C03641=1066.712,243.059,411.910,173.514,30.736,155.609
C03642=1066.719,243.308,411.883,173.516,30.739,155.610
C03643=1066.724,243.556,411.855,173.519,30.744,155.610
C03644=1066.731,243.805,411.827,173.521,30.748,155.611
C03645=1066.736,244.053,411.800,173.523,30.751,155.612
C03646=1066.743,244.302,411.772,173.526,30.756,155.613
C03647=1066.748,244.550,411.744,173.527,30.759,155.613
C03648=1066.754,244.799,411.717,173.530,30.763,155.614
C03649=1066.760,245.047,411.689,173.533,30.768,155.615
C03650=1066.766,245.295,411.661,173.534,30.771,155.615
C03651=1066.772,245.543,411.634,173.537,30.775,155.616
C03652=1066.778,245.792,411.606,173.540,30.780,155.617
C03653=1066.783,246.041,411.579,173.542,30.783,155.617
C03654=1066.790,246.289,411.551,173.544,30.787,155.618
C03655=1066.796,246.538,411.522,173.547,30.792,155.619
C03656=1066.802,246.785,411.495,173.549,30.795,155.619
C03657=1066.808,247.034,411.467,173.551,30.799,155.620
C03658=1066.813,247.283,411.440,173.553,30.804,155.621
C03659=1066.819,247.532,411.411,173.556,30.807,155.622
C03660=1066.825,247.779,411.384,173.558,30.812,155.622
C03661=1066.831,248.028,411.356,173.560,30.815,155.623
C03662=1066.836,248.276,411.328,173.563,30.819,155.624
C03663=1066.843,248.525,411.300,173.566,30.824,155.624
C03664=1066.848,248.740,411.275,173.567,30.827,155.625
C03665=1066.853,248.954,411.252,173.569,30.831,155.626
C03666=1066.858,249.169,411.227,173.572,30.834,155.626
C03667=1066.863,249.384,411.203,173.574,30.838,155.627
C03668=1066.868,249.599,411.179,173.575,30.841,155.627
C03669=1066.873,249.814,411.155,173.577,30.844,155.628
C03670=1066.878,250.029,411.130,173.580,30.848,155.629
C03671=1066.884,250.244,411.106,173.582,30.851,155.629
C03672=1066.889,250.492,411.078,173.584,30.855,155.630
C03673=1066.895,250.740,411.049,173.586,30.859,155.631
C03674=1066.901,250.989,411.021,173.589,30.863,155.631
C03675=1066.907,251.237,410.994,173.591,30.868,155.632
C03676=1066.913,251.485,410.965,173.593,30.871,155.633
C03677=1066.918,251.733,410.937,173.596,30.875,155.634
C03678=1066.924,251.982,410.909,173.599,30.880,155.634
C03679=1066.930,252.231,410.881,173.600,30.883,155.635
C03680=1066.936,252.479,410.853,173.603,30.887,155.636
C03681=1066.942,252.727,410.825,173.606,30.892,155.636
C03682=1066.949,252.976,410.796,173.608,30.896,155.637
C03683=1066.954,253.224,410.768,173.610,30.899,155.638
C03684=1066.961,253.472,410.740,173.613,30.904,155.639
C03685=1066.967,253.721,410.712,173.616,30.907,155.639
C03686=1066.972,253.969,410.684,173.617,30.911,155.640
C03687=1066.978,254.217,410.655,173.620,30.916,155.641
C03688=1066.984,254.466,410.627,173.623,30.919,155.641
C03689=1066.991,254.714,410.599,173.625,30.923,155.642
C03690=1066.996,254.962,410.571,173.627,30.927,155.643
C03691=1067.002,255.210,410.542,173.630,30.931,155.643
C03692=1067.008,255.459,410.514,173.633,30.935,155.644
C03693=1067.014,255.707,410.486,173.634,30.939,155.645
C03694=1067.020,255.955,410.457,173.637,30.943,155.645
C03695=1067.027,256.204,410.429,173.640,30.947,155.646
C03696=1067.033,256.453,410.401,173.642,30.951,155.647
C03697=1067.039,256.701,410.372,173.644,30.955,155.648
C03698=1067.044,256.949,410.344,173.647,30.959,155.648
C03699=1067.050,257.197,410.315,173.650,30.963,155.649
C03700=1067.056,257.446,410.286,173.652,30.967,155.650
C03701=1067.063,257.694,410.258,173.654,30.971,155.650
C03702=1067.069,257.941,410.230,173.657,30.975,155.651
C03703=1067.075,258.190,410.201,173.660,30.979,155.652
C03704=1067.081,258.439,410.173,173.661,30.983,155.652
C03705=1067.087,258.687,410.144,173.664,30.987,155.653
C03706=1067.093,258.936,410.116,173.667,30.991,155.654
C03707=1067.099,259.184,410.087,173.669,30.994,155.654
C03708=1067.104,259.432,410.059,173.672,30.999,155.655
C03709=1067.111,259.680,410.030,173.674,31.002,155.656
C03710=1067.117,259.929,410.002,173.677,31.006,155.657
C03711=1067.124,260.177,409.973,173.679,31.010,155.657
C03712=1067.130,260.425,409.944,173.682,31.015,155.658
C03713=1067.136,260.674,409.916,173.684,31.018,155.659
C03714=1067.142,260.922,409.887,173.687,31.022,155.659
C03715=1067.148,261.171,409.858,173.689,31.026,155.660
C03716=1067.154,261.419,409.829,173.692,31.030,155.661
C03717=1067.160,261.666,409.801,173.695,31.034,155.661
C03718=1067.167,261.914,409.773,173.697,31.038,155.662
C03719=1067.173,262.163,409.744,173.699,31.042,155.663
C03720=1067.178,262.377,409.719,173.701,31.045,155.663
C03721=1067.183,262.591,409.694,173.704,31.049,155.664
C03722=1067.189,262.805,409.670,173.706,31.052,155.665
C03723=1067.194,263.018,409.644,173.708,31.055,155.665
C03724=1067.199,263.232,409.620,173.710,31.059,155.666
C03725=1067.205,263.446,409.595,173.713,31.062,155.666
C03726=1067.210,263.659,409.571,173.715,31.066,155.667
C03727=1067.215,263.873,409.545,173.716,31.069,155.668
C03728=1067.221,264.121,409.517,173.719,31.073,155.668
C03729=1067.227,264.369,409.488,173.722,31.077,155.669
C03730=1067.232,264.618,409.458,173.725,31.081,155.670
C03731=1067.239,264.866,409.429,173.727,31.085,155.670
C03732=1067.245,265.114,409.400,173.729,31.089,155.671
C03733=1067.251,265.362,409.371,173.732,31.093,155.672
C03734=1067.256,265.611,409.342,173.735,31.097,155.673
C03735=1067.263,265.859,409.313,173.737,31.101,155.673
C03736=1067.269,266.108,409.284,173.740,31.105,155.674
C03737=1067.275,266.356,409.255,173.742,31.109,155.675
C03738=1067.281,266.604,409.225,173.745,31.113,155.675
C03739=1067.287,266.852,409.196,173.747,31.117,155.676
C03740=1067.293,267.100,409.167,173.750,31.121,155.677
C03741=1067.299,267.349,409.138,173.753,31.125,155.678
C03742=1067.305,267.597,409.109,173.755,31.129,155.678
C03743=1067.311,267.845,409.080,173.757,31.133,155.679
C03744=1067.317,268.093,409.051,173.760,31.137,155.680
C03745=1067.324,268.341,409.022,173.763,31.141,155.680
C03746=1067.329,268.590,408.992,173.766,31.145,155.681
C03747=1067.335,268.838,408.963,173.768,31.149,155.682
C03748=1067.342,269.086,408.934,173.771,31.153,155.682
C03749=1067.347,269.335,408.904,173.773,31.157,155.683
C03750=1067.353,269.583,408.875,173.776,31.161,155.684
C03751=1067.360,269.831,408.846,173.778,31.165,155.685
C03752=1067.365,270.079,408.816,173.781,31.169,155.685
C03753=1067.372,270.327,408.787,173.784,31.173,155.686
C03754=1067.377,270.575,408.757,173.787,31.177,155.687
C03755=1067.383,270.823,408.728,173.788,31.181,155.687
C03756=1067.390,271.071,408.699,173.791,31.185,155.688
C03757=1067.395,271.320,408.669,173.794,31.189,155.689
C03758=1067.401,271.568,408.640,173.797,31.193,155.690
C03759=1067.407,271.816,408.610,173.799,31.197,155.690
C03760=1067.414,272.064,408.581,173.802,31.201,155.691
C03761=1067.419,272.312,408.551,173.805,31.205,155.692
C03762=1067.425,272.561,408.522,173.807,31.209,155.692
C03763=1067.431,272.808,408.492,173.809,31.213,155.693
C03764=1067.437,273.057,408.463,173.812,31.217,155.694
C03765=1067.443,273.306,408.433,173.815,31.221,155.695
C03766=1067.450,273.553,408.403,173.818,31.225,155.695
C03767=1067.456,273.802,408.373,173.820,31.229,155.696
C03768=1067.462,274.050,408.344,173.823,31.234,155.697
C03769=1067.468,274.298,408.314,173.826,31.237,155.697
C03770=1067.474,274.546,408.285,173.829,31.242,155.698
C03771=1067.480,274.794,408.255,173.830,31.245,155.699
C03772=1067.485,275.042,408.225,173.833,31.249,155.700
C03773=1067.491,275.290,408.196,173.836,31.254,155.700
C03774=1067.498,275.539,408.165,173.839,31.257,155.701
C03775=1067.504,275.787,408.136,173.841,31.262,155.702
C03776=1067.509,276.002,408.110,173.844,31.265,155.702
C03777=1067.515,276.218,408.084,173.846,31.269,155.703
C03778=1067.520,276.433,408.058,173.849,31.272,155.704
C03779=1067.525,276.649,408.032,173.851,31.275,155.704
C03780=1067.530,276.864,408.006,173.853,31.279,155.705
C03781=1067.535,277.080,407.980,173.855,31.283,155.706
C03782=1067.541,277.295,407.955,173.858,31.286,155.706
C03783=1067.546,277.510,407.928,173.860,31.290,155.707
C03784=1067.551,277.759,407.899,173.862,31.294,155.708
C03785=1067.558,278.006,407.869,173.865,31.298,155.708
C03786=1067.564,278.255,407.838,173.868,31.302,155.709
C03787=1067.570,278.503,407.809,173.871,31.306,155.710
C03788=1067.576,278.751,407.778,173.874,31.310,155.710
C03789=1067.582,278.999,407.749,173.876,31.314,155.711
C03790=1067.588,279.247,407.719,173.879,31.318,155.712
C03791=1067.594,279.496,407.688,173.882,31.322,155.713
C03792=1067.600,279.744,407.659,173.885,31.326,155.713
C03793=1067.606,279.992,407.629,173.887,31.331,155.714
C03794=1067.612,280.239,407.598,173.889,31.334,155.715
C03795=1067.618,280.488,407.568,173.892,31.339,155.716
C03796=1067.625,280.736,407.539,173.895,31.342,155.716
C03797=1067.631,280.984,407.508,173.897,31.347,155.717
C03798=1067.636,281.232,407.478,173.900,31.351,155.718
C03799=1067.643,281.480,407.447,173.903,31.355,155.718
C03800=1067.649,281.728,407.417,173.906,31.359,155.719
C03801=1067.654,281.976,407.387,173.908,31.363,155.720
C03802=1067.660,282.224,407.357,173.911,31.367,155.721
C03803=1067.666,282.473,407.326,173.914,31.372,155.722
C03804=1067.672,282.721,407.296,173.917,31.375,155.722
C03805=1067.678,282.968,407.266,173.920,31.380,155.723
C03806=1067.684,283.216,407.235,173.922,31.384,155.724
C03807=1067.691,283.464,407.205,173.925,31.388,155.724
C03808=1067.697,283.712,407.175,173.928,31.392,155.725
C03809=1067.703,283.960,407.144,173.931,31.396,155.726
C03810=1067.709,284.209,407.114,173.933,31.400,155.727
C03811=1067.715,284.457,407.084,173.936,31.404,155.727
C03812=1067.720,284.705,407.054,173.939,31.408,155.728
C03813=1067.727,284.953,407.022,173.942,31.412,155.729
C03814=1067.733,285.201,406.992,173.945,31.417,155.730
C03815=1067.739,285.448,406.962,173.947,31.421,155.730
C03816=1067.745,285.697,406.931,173.950,31.425,155.731
C03817=1067.751,285.945,406.900,173.953,31.429,155.732
C03818=1067.757,286.193,406.870,173.956,31.433,155.732
C03819=1067.763,286.441,406.839,173.958,31.437,155.733
C03820=1067.769,286.689,406.809,173.961,31.441,155.734
C03821=1067.775,286.938,406.778,173.964,31.445,155.735
C03822=1067.781,287.185,406.748,173.967,31.450,155.736
C03823=1067.788,287.434,406.717,173.970,31.453,155.736
C03824=1067.794,287.681,406.686,173.972,31.458,155.737
C03825=1067.800,287.929,406.656,173.975,31.462,155.738
C03826=1067.806,288.177,406.625,173.978,31.466,155.738
C03827=1067.812,288.425,406.595,173.981,31.470,155.739
C03828=1067.818,288.674,406.564,173.983,31.474,155.740
C03829=1067.824,288.921,406.533,173.986,31.478,155.741
C03830=1067.831,289.169,406.502,173.989,31.482,155.741
C03831=1067.837,289.417,406.472,173.992,31.486,155.742
C03832=1067.842,289.635,406.445,173.995,31.490,155.743
C03833=1067.847,289.853,406.418,173.996,31.494,155.744
C03834=1067.852,290.070,406.391,173.999,31.497,155.744
C03835=1067.858,290.288,406.363,174.002,31.501,155.745
C03836=1067.863,290.506,406.336,174.004,31.505,155.746
C03837=1067.868,290.724,406.309,174.007,31.509,155.746
C03838=1067.874,290.942,406.282,174.009,31.512,155.747
C03839=1067.879,291.160,406.255,174.011,31.515,155.747
C03840=1067.885,291.408,406.224,174.014,31.520,155.748
C03841=1067.891,291.655,406.193,174.017,31.524,155.749
C03842=1067.897,291.904,406.162,174.021,31.528,155.750
C03843=1067.903,292.151,406.131,174.023,31.532,155.750
C03844=1067.910,292.400,406.100,174.026,31.537,155.751
C03845=1067.916,292.647,406.069,174.029,31.541,155.752
C03846=1067.921,292.896,406.038,174.032,31.545,155.753
C03847=1067.928,293.143,406.007,174.035,31.549,155.754
C03848=1067.934,293.392,405.976,174.037,31.553,155.754
C03849=1067.939,293.639,405.944,174.040,31.558,155.755
C03850=1067.946,293.888,405.913,174.043,31.561,155.756
C03851=1067.952,294.135,405.882,174.046,31.566,155.757
C03852=1067.959,294.383,405.851,174.049,31.570,155.757
C03853=1067.964,294.632,405.820,174.051,31.574,155.758
C03854=1067.970,294.879,405.789,174.054,31.579,155.759
C03855=1067.977,295.127,405.758,174.058,31.582,155.760
C03856=1067.982,295.375,405.726,174.061,31.587,155.760
C03857=1067.989,295.623,405.695,174.064,31.591,155.761
C03858=1067.995,295.871,405.664,174.066,31.595,155.762
C03859=1068.001,296.119,405.632,174.069,31.600,155.763
C03860=1068.007,296.367,405.601,174.072,31.603,155.763
C03861=1068.013,296.614,405.569,174.075,31.608,155.764
C03862=1068.019,296.863,405.539,174.078,31.612,155.765
C03863=1068.025,297.110,405.507,174.080,31.616,155.766
C03864=1068.031,297.358,405.475,174.083,31.621,155.767
C03865=1068.037,297.606,405.443,174.087,31.625,155.767
C03866=1068.043,297.854,405.412,174.090,31.629,155.768
C03867=1068.049,298.102,405.381,174.093,31.634,155.769
C03868=1068.055,298.350,405.349,174.095,31.638,155.770
C03869=1068.061,298.598,405.318,174.098,31.642,155.771
C03870=1068.067,298.845,405.286,174.101,31.647,155.771
C03871=1068.073,299.094,405.254,174.104,31.651,155.772
C03872=1068.079,299.341,405.223,174.107,31.655,155.773
C03873=1068.085,299.589,405.191,174.109,31.659,155.774
C03874=1068.091,299.837,405.159,174.113,31.664,155.775
C03875=1068.097,300.085,405.128,174.116,31.668,155.775
C03876=1068.103,300.339,405.095,174.119,31.673,155.776
C03877=1068.109,300.592,405.063,174.122,31.677,155.777
C03878=1068.115,300.846,405.030,174.124,31.681,155.778
C03879=1068.121,301.099,404.998,174.128,31.686,155.779
C03880=1068.127,301.348,404.966,174.131,31.690,155.779
C03881=1068.134,301.595,404.934,174.134,31.694,155.780
C03882=1068.139,301.843,404.902,174.137,31.698,155.781
C03883=1068.145,302.091,404.870,174.139,31.703,155.782
C03884=1068.152,302.338,404.839,174.142,31.708,155.783
C03885=1068.158,302.587,404.807,174.146,31.712,155.783
C03886=1068.164,302.835,404.775,174.149,31.716,155.784
C03887=1068.170,303.083,404.743,174.152,31.721,155.785
C03888=1068.175,303.310,404.714,174.154,31.724,155.786
C03889=1068.181,303.538,404.685,174.157,31.729,155.786
C03890=1068.186,303.767,404.655,174.160,31.732,155.787
C03891=1068.193,303.995,404.626,174.163,31.737,155.788
C03892=1068.197,304.223,404.596,174.166,31.740,155.789
C03893=1068.203,304.452,404.567,174.168,31.744,155.789
C03894=1068.209,304.679,404.538,174.170,31.748,155.790
C03895=1068.214,304.908,404.508,174.173,31.752,155.791
C03896=1068.221,305.156,404.475,174.177,31.757,155.792
C03897=1068.227,305.403,404.444,174.180,31.761,155.792
C03898=1068.233,305.651,404.412,174.183,31.765,155.793
C03899=1068.239,305.899,404.379,174.185,31.770,155.794
C03900=1068.245,306.147,404.347,174.188,31.774,155.795
C03901=1068.252,306.395,404.316,174.192,31.778,155.796
C03902=1068.257,306.642,404.284,174.195,31.783,155.796
C03903=1068.263,306.890,404.252,174.198,31.787,155.797
C03904=1068.270,307.137,404.219,174.201,31.791,155.798
C03905=1068.276,307.386,404.187,174.203,31.796,155.799
C03906=1068.282,307.634,404.155,174.207,31.800,155.800
C03907=1068.289,307.881,404.123,174.210,31.805,155.801
C03908=1068.295,308.129,404.091,174.213,31.809,155.801
C03909=1068.301,308.377,404.058,174.216,31.813,155.802
C03910=1068.307,308.625,404.026,174.220,31.818,155.803
C03911=1068.313,308.873,403.993,174.222,31.822,155.804
C03912=1068.319,309.120,403.961,174.225,31.826,155.805
C03913=1068.326,309.367,403.929,174.228,31.831,155.805
C03914=1068.332,309.616,403.897,174.232,31.835,155.806
C03915=1068.338,309.863,403.865,174.235,31.839,155.807
C03916=1068.344,310.111,403.832,174.237,31.844,155.808
C03917=1068.350,310.359,403.800,174.240,31.848,155.809
C03918=1068.357,310.607,403.767,174.244,31.853,155.809
C03919=1068.363,310.854,403.734,174.247,31.857,155.810
C03920=1068.370,311.102,403.703,174.250,31.861,155.811
C03921=1068.376,311.350,403.670,174.254,31.866,155.812
C03922=1068.382,311.597,403.637,174.256,31.870,155.813
C03923=1068.388,311.846,403.605,174.259,31.875,155.814
C03924=1068.394,312.093,403.573,174.262,31.879,155.814
C03925=1068.401,312.341,403.540,174.266,31.883,155.815
C03926=1068.407,312.590,403.507,174.269,31.888,155.816
C03927=1068.414,312.837,403.475,174.272,31.892,155.817
C03928=1068.420,313.085,403.442,174.275,31.896,155.818
C03929=1068.426,313.332,403.409,174.278,31.901,155.818
C03930=1068.433,313.580,403.377,174.281,31.905,155.819
C03931=1068.439,313.828,403.345,174.284,31.910,155.820
C03932=1068.446,314.076,403.312,174.288,31.914,155.821
C03933=1068.451,314.323,403.279,174.291,31.919,155.822
C03934=1068.457,314.571,403.246,174.293,31.923,155.823
C03935=1068.464,314.819,403.213,174.297,31.928,155.824
C03936=1068.469,315.067,403.180,174.300,31.932,155.824
C03937=1068.476,315.314,403.147,174.303,31.937,155.825
C03938=1068.482,315.562,403.115,174.306,31.941,155.826
C03939=1068.487,315.810,403.081,174.310,31.946,155.827
C03940=1068.494,316.057,403.049,174.312,31.951,155.828
C03941=1068.499,316.305,403.015,174.315,31.955,155.829
C03942=1068.506,316.553,402.982,174.319,31.960,155.829
C03943=1068.512,316.800,402.950,174.322,31.965,155.830
C03944=1068.518,317.031,402.919,174.325,31.969,155.831
C03945=1068.523,317.261,402.888,174.328,31.973,155.832
C03946=1068.529,317.490,402.858,174.331,31.977,155.833
C03947=1068.535,317.721,402.826,174.333,31.982,155.834
C03948=1068.540,317.951,402.796,174.336,31.986,155.834
C03949=1068.545,318.180,402.765,174.339,31.990,155.835
C03950=1068.552,318.411,402.734,174.343,31.994,155.836
C03951=1068.557,318.640,402.703,174.346,31.999,155.837
C03952=1068.564,318.888,402.670,174.349,32.003,155.838
C03953=1068.569,319.135,402.637,174.352,32.008,155.839
C03954=1068.575,319.383,402.604,174.355,32.013,155.839
C03955=1068.582,319.631,402.570,174.358,32.017,155.840
C03956=1068.588,319.879,402.537,174.361,32.022,155.841
C03957=1068.594,320.127,402.504,174.365,32.027,155.842
C03958=1068.600,320.374,402.471,174.368,32.031,155.843
C03959=1068.606,320.621,402.437,174.371,32.036,155.844
C03960=1068.613,320.870,402.404,174.374,32.040,155.845
C03961=1068.618,321.118,402.371,174.377,32.045,155.846
C03962=1068.625,321.365,402.337,174.380,32.049,155.847
C03963=1068.630,321.613,402.304,174.384,32.054,155.847
C03964=1068.638,321.860,402.270,174.387,32.059,155.848
C03965=1068.643,322.108,402.237,174.391,32.064,155.849
C03966=1068.649,322.356,402.204,174.394,32.068,155.850
C03967=1068.655,322.603,402.170,174.396,32.073,155.851
C03968=1068.662,322.851,402.137,174.400,32.077,155.852
C03969=1068.668,323.099,402.103,174.403,32.082,155.853
C03970=1068.674,323.346,402.070,174.407,32.087,155.854
C03971=1068.681,323.594,402.036,174.410,32.091,155.854
C03972=1068.687,323.842,402.003,174.413,32.096,155.855
C03973=1068.693,324.089,401.969,174.417,32.101,155.856
C03974=1068.700,324.337,401.936,174.419,32.105,155.857
C03975=1068.706,324.585,401.902,174.423,32.110,155.858
C03976=1068.712,324.832,401.869,174.426,32.115,155.859
C03977=1068.718,325.080,401.834,174.429,32.119,155.860
C03978=1068.724,325.327,401.800,174.433,32.124,155.861
C03979=1068.731,325.576,401.767,174.436,32.129,155.862
C03980=1068.737,325.823,401.733,174.440,32.134,155.863
C03981=1068.744,326.070,401.700,174.442,32.138,155.863
C03982=1068.750,326.319,401.666,174.446,32.143,155.864
C03983=1068.756,326.566,401.633,174.449,32.148,155.865
C03984=1068.763,326.814,401.598,174.452,32.152,155.866
C03985=1068.768,327.061,401.565,174.456,32.157,155.867
C03986=1068.776,327.309,401.531,174.459,32.162,155.868
C03987=1068.782,327.556,401.497,174.463,32.166,155.869
C03988=1068.789,327.804,401.463,174.466,32.171,155.870
C03989=1068.795,328.051,401.429,174.469,32.176,155.871
C03990=1068.801,328.300,401.395,174.472,32.181,155.872
C03991=1068.807,328.547,401.362,174.476,32.186,155.872
C03992=1068.814,328.795,401.327,174.479,32.190,155.873
C03993=1068.820,329.042,401.294,174.483,32.195,155.874
C03994=1068.827,329.290,401.260,174.486,32.200,155.875
C03995=1068.833,329.537,401.226,174.490,32.204,155.876
C03996=1068.840,329.785,401.192,174.493,32.209,155.877
C03997=1068.846,330.032,401.158,174.496,32.214,155.878
C03998=1068.852,330.280,401.123,174.499,32.219,155.879
C03999=1068.859,330.528,401.089,174.503,32.224,155.880
C04000=1068.865,330.755,401.059,174.506,32.228,155.881
C04001=1068.871,330.982,401.027,174.509,32.232,155.881
C04002=1068.876,331.209,400.996,174.512,32.237,155.882
C04003=1068.882,331.435,400.965,174.515,32.241,155.883
C04004=1068.888,331.662,400.933,174.519,32.246,155.884
C04005=1068.894,331.889,400.902,174.521,32.250,155.885
C04006=1068.900,332.116,400.871,174.524,32.255,155.886
C04007=1068.905,332.343,400.839,174.527,32.259,155.887
C04008=1068.912,332.590,400.804,174.531,32.264,155.888
C04009=1068.918,332.838,400.770,174.534,32.269,155.888
C04010=1068.924,333.086,400.736,174.538,32.274,155.890
C04011=1068.930,333.333,400.702,174.541,32.279,155.890
C04012=1068.937,333.581,400.667,174.545,32.284,155.891
C04013=1068.943,333.828,400.632,174.548,32.289,155.892
C04014=1068.949,334.075,400.598,174.551,32.294,155.893
C04015=1068.956,334.323,400.564,174.554,32.299,155.894
C04016=1068.962,334.571,400.530,174.558,32.304,155.895
C04017=1068.968,334.818,400.495,174.562,32.308,155.896
C04018=1068.975,335.066,400.460,174.565,32.314,155.897
C04019=1068.981,335.313,400.426,174.569,32.319,155.898
C04020=1068.987,335.561,400.390,174.572,32.323,155.899
C04021=1068.993,335.809,400.356,174.576,32.329,155.900
C04022=1068.999,336.056,400.321,174.579,32.333,155.901
C04023=1069.006,336.304,400.287,174.582,32.338,155.902
C04024=1069.012,336.552,400.252,174.585,32.344,155.903
C04025=1069.019,336.799,400.217,174.589,32.348,155.904
C04026=1069.025,337.046,400.183,174.593,32.353,155.905
C04027=1069.032,337.294,400.148,174.596,32.359,155.906
C04028=1069.038,337.542,400.114,174.600,32.363,155.907
C04029=1069.044,337.788,400.079,174.603,32.369,155.908
C04030=1069.051,338.036,400.044,174.607,32.374,155.909
C04031=1069.057,338.284,400.009,174.611,32.379,155.910
C04032=1069.064,338.531,399.973,174.614,32.384,155.911
C04033=1069.069,338.779,399.939,174.617,32.389,155.912
C04034=1069.075,339.026,399.904,174.620,32.394,155.913
C04035=1069.082,339.274,399.869,174.624,32.399,155.914
C04036=1069.088,339.521,399.835,174.628,32.404,155.915
C04037=1069.095,339.768,399.799,174.631,32.409,155.916
C04038=1069.101,340.016,399.764,174.635,32.415,155.917
C04039=1069.107,340.264,399.729,174.638,32.419,155.918
C04040=1069.114,340.511,399.694,174.642,32.425,155.919
C04041=1069.120,340.758,399.659,174.646,32.430,155.920
C04042=1069.126,341.006,399.624,174.649,32.435,155.921
C04043=1069.133,341.254,399.589,174.653,32.440,155.922
C04044=1069.140,341.501,399.554,174.655,32.445,155.923
C04045=1069.146,341.749,399.518,174.659,32.450,155.924
C04046=1069.152,341.996,399.483,174.663,32.456,155.925
C04047=1069.159,342.243,399.448,174.666,32.461,155.926
C04048=1069.165,342.490,399.413,174.670,32.466,155.927
C04049=1069.171,342.738,399.378,174.674,32.471,155.928
C04050=1069.178,342.985,399.342,174.677,32.476,155.929
C04051=1069.184,343.233,399.307,174.681,32.481,155.930
C04052=1069.191,343.481,399.272,174.685,32.487,155.931
C04053=1069.197,343.728,399.237,174.688,32.492,155.932
C04054=1069.203,343.976,399.201,174.692,32.497,155.933
C04055=1069.210,344.223,399.166,174.696,32.503,155.934
C04056=1069.216,344.448,399.134,174.699,32.507,155.935
C04057=1069.221,344.672,399.102,174.701,32.512,155.936
C04058=1069.228,344.896,399.070,174.705,32.517,155.937
C04059=1069.233,345.121,399.037,174.708,32.522,155.938
C04060=1069.239,345.345,399.005,174.711,32.526,155.939
C04061=1069.244,345.570,398.973,174.715,32.531,155.940
C04062=1069.251,345.793,398.940,174.718,32.536,155.941
C04063=1069.257,346.018,398.908,174.722,32.541,155.942
C04064=1069.263,346.266,398.872,174.725,32.546,155.943
C04065=1069.269,346.512,398.837,174.729,32.552,155.944
C04066=1069.275,346.760,398.802,174.733,32.557,155.945
C04067=1069.282,347.007,398.766,174.736,32.562,155.946
C04068=1069.288,347.254,398.730,174.740,32.568,155.947
C04069=1069.294,347.502,398.694,174.744,32.573,155.948
C04070=1069.301,347.749,398.659,174.747,32.578,155.949
C04071=1069.307,347.996,398.623,174.751,32.584,155.950
C04072=1069.313,348.244,398.587,174.754,32.589,155.952
C04073=1069.320,348.492,398.552,174.758,32.594,155.953
C04074=1069.327,348.739,398.515,174.761,32.600,155.954
C04075=1069.333,348.987,398.479,174.765,32.605,155.955
C04076=1069.340,349.234,398.443,174.769,32.611,155.956
C04077=1069.346,349.481,398.408,174.773,32.616,155.957
C04078=1069.352,349.728,398.371,174.776,32.622,155.958
C04079=1069.359,349.976,398.336,174.780,32.627,155.959
C04080=1069.365,350.223,398.300,174.784,32.633,155.960
C04081=1069.371,350.470,398.264,174.788,32.638,155.961
C04082=1069.379,350.717,398.228,174.791,32.644,155.963
C04083=1069.385,350.965,398.192,174.795,32.649,155.964
C04084=1069.391,351.212,398.156,174.799,32.654,155.965
C04085=1069.399,351.459,398.120,174.803,32.660,155.966
C04086=1069.405,351.707,398.084,174.807,32.666,155.967
C04087=1069.411,351.954,398.048,174.810,32.671,155.968
C04088=1069.417,352.202,398.012,174.814,32.677,155.969
C04089=1069.423,352.449,397.975,174.818,32.682,155.970
C04090=1069.430,352.696,397.940,174.822,32.688,155.971
C04091=1069.437,352.943,397.903,174.826,32.693,155.972
C04092=1069.443,353.191,397.867,174.828,32.699,155.974
C04093=1069.450,353.438,397.831,174.832,32.704,155.975
C04094=1069.456,353.685,397.794,174.836,32.710,155.976
C04095=1069.462,353.932,397.758,174.840,32.716,155.977
C04096=1069.469,354.179,397.721,174.844,32.721,155.978
C04097=1069.476,354.427,397.684,174.847,32.727,155.979
C04098=1069.482,354.675,397.649,174.851,32.732,155.980
C04099=1069.488,354.922,397.612,174.855,32.738,155.982
C04100=1069.494,355.169,397.576,174.859,32.744,155.983
C04101=1069.501,355.416,397.539,174.863,32.750,155.984
C04102=1069.508,355.664,397.503,174.867,32.755,155.985
C04103=1069.515,355.910,397.467,174.870,32.761,155.986
C04104=1069.521,356.157,397.430,174.874,32.766,155.987
C04105=1069.527,356.404,397.394,174.878,32.772,155.988
C04106=1069.534,356.652,397.357,174.882,32.778,155.990
C04107=1069.541,356.899,397.321,174.886,32.784,155.991
C04108=1069.547,357.146,397.284,174.890,32.790,155.992
C04109=1069.554,357.393,397.247,174.894,32.795,155.993
C04110=1069.561,357.641,397.210,174.898,32.801,155.994
C04111=1069.567,357.888,397.174,174.901,32.807,155.995
C04112=1069.573,358.114,397.140,174.905,32.812,155.997
C04113=1069.579,358.340,397.106,174.909,32.817,155.998
C04114=1069.585,358.566,397.073,174.912,32.823,155.999
C04115=1069.591,358.793,397.039,174.916,32.828,156.000
C04116=1069.597,359.019,397.005,174.919,32.833,156.001
C04117=1069.603,359.245,396.972,174.923,32.839,156.002
C04118=1069.608,359.472,396.937,174.926,32.844,156.003
C04119=1069.615,359.698,396.904,174.930,32.849,156.004
C04120=1069.621,359.946,396.867,174.934,32.855,156.005
C04121=1069.628,360.193,396.830,174.938,32.861,156.007
C04122=1069.635,360.440,396.793,174.942,32.867,156.008
C04123=1069.641,360.687,396.756,174.946,32.873,156.009
C04124=1069.647,360.934,396.719,174.950,32.879,156.010
C04125=1069.654,361.181,396.682,174.953,32.885,156.011
C04126=1069.661,361.428,396.645,174.957,32.891,156.013
C04127=1069.668,361.675,396.608,174.961,32.896,156.014
C04128=1069.674,361.923,396.571,174.965,32.902,156.015
C04129=1069.681,362.170,396.533,174.969,32.909,156.016
C04130=1069.687,362.417,396.497,174.973,32.914,156.018
C04131=1069.694,362.664,396.459,174.977,32.920,156.019
C04132=1069.701,362.911,396.422,174.981,32.926,156.020
C04133=1069.707,363.159,396.385,174.985,32.932,156.021
C04134=1069.714,363.405,396.348,174.989,32.938,156.022
C04135=1069.721,363.653,396.311,174.993,32.945,156.024
C04136=1069.727,363.899,396.274,174.997,32.950,156.025
C04137=1069.734,364.147,396.235,175.001,32.956,156.026
C04138=1069.740,364.393,396.198,175.005,32.963,156.028
C04139=1069.747,364.641,396.162,175.009,32.968,156.029
C04140=1069.753,364.888,396.124,175.013,32.975,156.030
C04141=1069.761,365.135,396.086,175.017,32.980,156.031
C04142=1069.766,365.382,396.048,175.021,32.987,156.033
C04143=1069.774,365.629,396.011,175.025,32.993,156.034
C04144=1069.779,365.876,395.974,175.029,32.999,156.035
C04145=1069.787,366.123,395.936,175.033,33.005,156.036
C04146=1069.793,366.371,395.898,175.037,33.012,156.038
C04147=1069.800,366.617,395.861,175.041,33.018,156.039
C04148=1069.806,366.864,395.823,175.045,33.024,156.040
C04149=1069.813,367.111,395.786,175.049,33.030,156.042
C04150=1069.819,367.358,395.748,175.053,33.036,156.043
C04151=1069.827,367.606,395.710,175.058,33.043,156.044
C04152=1069.832,367.852,395.672,175.062,33.049,156.046
C04153=1069.839,368.100,395.634,175.066,33.055,156.047
C04154=1069.846,368.346,395.597,175.070,33.061,156.048
C04155=1069.852,368.594,395.559,175.074,33.068,156.049
C04156=1069.860,368.840,395.521,175.078,33.074,156.051
C04157=1069.866,369.087,395.483,175.082,33.080,156.052
C04158=1069.873,369.334,395.445,175.086,33.087,156.053
C04159=1069.879,369.581,395.407,175.090,33.093,156.055
C04160=1069.887,369.829,395.370,175.094,33.099,156.056
C04161=1069.893,370.075,395.331,175.099,33.106,156.057
C04162=1069.899,370.322,395.293,175.103,33.112,156.059
C04163=1069.907,370.569,395.256,175.107,33.118,156.060
C04164=1069.913,370.817,395.218,175.111,33.125,156.061
C04165=1069.920,371.062,395.180,175.115,33.131,156.063
C04166=1069.926,371.310,395.142,175.119,33.138,156.064
C04167=1069.933,371.557,395.103,175.123,33.144,156.065
C04168=1069.939,371.792,395.067,175.127,33.150,156.067
C04169=1069.946,372.026,395.030,175.132,33.156,156.068
C04170=1069.953,372.262,394.995,175.136,33.162,156.069
C04171=1069.959,372.496,394.958,175.140,33.168,156.071
C04172=1069.966,372.730,394.922,175.144,33.174,156.072
C04173=1069.972,372.966,394.886,175.148,33.181,156.073
C04174=1069.979,373.200,394.849,175.152,33.187,156.074
C04175=1069.984,373.435,394.812,175.155,33.193,156.076
C04176=1069.992,373.682,394.775,175.160,33.200,156.077
C04177=1069.999,373.929,394.736,175.164,33.206,156.079
C04178=1070.005,374.176,394.698,175.168,33.213,156.080
C04179=1070.012,374.423,394.659,175.172,33.220,156.081
C04180=1070.018,374.669,394.620,175.176,33.226,156.083
C04181=1070.025,374.917,394.582,175.181,33.233,156.084
C04182=1070.031,375.164,394.544,175.186,33.240,156.086
C04183=1070.038,375.410,394.505,175.190,33.246,156.087
C04184=1070.045,375.657,394.466,175.194,33.253,156.088
C04185=1070.052,375.904,394.427,175.198,33.260,156.090
C04186=1070.058,376.152,394.389,175.202,33.266,156.091
C04187=1070.066,376.398,394.351,175.206,33.273,156.093
C04188=1070.073,376.645,394.312,175.211,33.280,156.094
C04189=1070.079,376.892,394.273,175.215,33.286,156.096
C04190=1070.086,377.138,394.234,175.220,33.293,156.097
C04191=1070.093,377.385,394.196,175.224,33.300,156.099
C04192=1070.099,377.631,394.157,175.228,33.307,156.100
C04193=1070.106,377.878,394.118,175.233,33.314,156.101
C04194=1070.113,378.125,394.079,175.237,33.320,156.103
C04195=1070.120,378.372,394.040,175.241,33.327,156.104
C04196=1070.127,378.619,394.001,175.245,33.334,156.106
C04197=1070.133,378.866,393.963,175.250,33.341,156.107
C04198=1070.141,379.113,393.923,175.255,33.348,156.109
C04199=1070.148,379.360,393.885,175.259,33.355,156.110
C04200=1070.154,379.607,393.846,175.263,33.361,156.112
C04201=1070.161,379.854,393.807,175.268,33.368,156.113
C04202=1070.168,380.100,393.767,175.272,33.375,156.115
C04203=1070.175,380.347,393.729,175.276,33.382,156.116
C04204=1070.182,380.593,393.690,175.280,33.389,156.118
C04205=1070.189,380.840,393.651,175.286,33.396,156.119
C04206=1070.196,381.086,393.611,175.290,33.403,156.121
C04207=1070.203,381.334,393.572,175.294,33.410,156.122
C04208=1070.210,381.581,393.533,175.299,33.417,156.124
C04209=1070.217,381.827,393.493,175.303,33.424,156.125
C04210=1070.223,382.074,393.454,175.307,33.431,156.127
C04211=1070.230,382.320,393.415,175.311,33.438,156.128
C04212=1070.237,382.567,393.375,175.317,33.445,156.130
C04213=1070.243,382.814,393.336,175.321,33.453,156.131
C04214=1070.250,383.061,393.297,175.325,33.459,156.133
C04215=1070.257,383.308,393.256,175.330,33.467,156.134
C04216=1070.264,383.555,393.218,175.334,33.474,156.136
C04217=1070.271,383.801,393.178,175.338,33.481,156.137
C04218=1070.277,384.048,393.139,175.344,33.488,156.139
C04219=1070.285,384.294,393.099,175.348,33.495,156.141
C04220=1070.292,384.540,393.059,175.352,33.503,156.142
C04221=1070.298,384.788,393.020,175.357,33.510,156.144
C04222=1070.305,385.034,392.980,175.361,33.517,156.145
C04223=1070.313,385.281,392.941,175.366,33.525,156.147
C04224=1070.319,385.534,392.900,175.371,33.532,156.149
C04225=1070.326,385.786,392.859,175.375,33.539,156.150
C04226=1070.334,386.039,392.819,175.380,33.547,156.152
C04227=1070.341,386.291,392.778,175.384,33.554,156.154
C04228=1070.348,386.537,392.738,175.390,33.562,156.155
C04229=1070.355,386.785,392.698,175.394,33.569,156.157
C04230=1070.362,387.031,392.658,175.399,33.577,156.158
C04231=1070.368,387.278,392.619,175.403,33.584,156.160
C04232=1070.376,387.525,392.579,175.408,33.592,156.162
C04233=1070.383,387.771,392.539,175.413,33.599,156.163
C04234=1070.389,388.018,392.499,175.417,33.606,156.165
C04235=1070.397,388.264,392.459,175.422,33.614,156.166
C04236=1070.404,388.510,392.418,175.426,33.621,156.168
C04237=1070.412,388.757,392.378,175.432,33.629,156.170
C04238=1070.419,389.003,392.339,175.436,33.636,156.171
C04239=1070.426,389.251,392.298,175.440,33.644,156.173
C04240=1070.433,389.497,392.259,175.445,33.651,156.175
C04241=1070.440,389.744,392.218,175.450,33.659,156.176
C04242=1070.447,389.990,392.179,175.455,33.666,156.178
C04243=1070.454,390.237,392.137,175.459,33.674,156.180
C04244=1070.461,390.483,392.098,175.464,33.681,156.181
C04245=1070.468,390.730,392.057,175.469,33.689,156.183
C04246=1070.475,390.977,392.018,175.474,33.697,156.185
C04247=1070.483,391.223,391.977,175.478,33.704,156.186
C04248=1070.489,391.470,391.936,175.483,33.712,156.188
C04249=1070.497,391.717,391.897,175.488,33.720,156.190
C04250=1070.503,391.962,391.856,175.493,33.728,156.192
C04251=1070.510,392.210,391.815,175.497,33.735,156.193
C04252=1070.518,392.455,391.775,175.502,33.743,156.195
C04253=1070.525,392.702,391.734,175.508,33.751,156.197
C04254=1070.532,392.948,391.694,175.512,33.759,156.198
C04255=1070.539,393.195,391.654,175.517,33.767,156.200
C04256=1070.547,393.442,391.612,175.522,33.775,156.202
C04257=1070.553,393.688,391.572,175.527,33.782,156.204
C04258=1070.560,393.935,391.531,175.531,33.791,156.206
C04259=1070.568,394.181,391.490,175.537,33.798,156.207
C04260=1070.575,394.427,391.450,175.541,33.806,156.209
C04261=1070.582,394.674,391.409,175.546,33.815,156.211
C04262=1070.589,394.921,391.368,175.551,33.822,156.213
C04263=1070.596,395.167,391.327,175.556,33.831,156.214
C04264=1070.603,395.413,391.286,175.561,33.838,156.216
C04265=1070.610,395.661,391.245,175.565,33.847,156.218
C04266=1070.617,395.907,391.204,175.571,33.855,156.220
C04267=1070.624,396.153,391.163,175.576,33.863,156.222
C04268=1070.632,396.399,391.122,175.580,33.871,156.223
C04269=1070.639,396.646,391.081,175.586,33.879,156.225
C04270=1070.647,396.893,391.040,175.590,33.887,156.227
C04271=1070.653,397.138,390.999,175.595,33.895,156.229
C04272=1070.661,397.385,390.958,175.601,33.903,156.231
C04273=1070.668,397.632,390.917,175.605,33.912,156.233
C04274=1070.675,397.878,390.875,175.610,33.920,156.234
C04275=1070.683,398.125,390.834,175.616,33.928,156.236
C04276=1070.690,398.371,390.793,175.620,33.937,156.238
C04277=1070.697,398.617,390.752,175.626,33.945,156.240
C04278=1070.704,398.864,390.711,175.631,33.953,156.242
C04279=1070.711,399.111,390.670,175.635,33.961,156.244
C04280=1070.719,399.378,390.624,175.641,33.971,156.246
C04281=1070.727,399.648,390.579,175.646,33.980,156.248
C04282=1070.734,399.916,390.534,175.653,33.989,156.250
C04283=1070.743,400.183,390.489,175.658,33.998,156.252
C04284=1070.749,400.430,390.447,175.662,34.007,156.254
C04285=1070.757,400.676,390.405,175.668,34.015,156.256
C04286=1070.764,400.923,390.364,175.673,34.024,156.258
C04287=1070.772,401.170,390.322,175.679,34.032,156.260
C04288=1070.779,401.415,390.280,175.683,34.041,156.262
C04289=1070.786,401.662,390.239,175.688,34.049,156.264
C04290=1070.793,401.908,390.197,175.694,34.058,156.266
C04291=1070.801,402.155,390.155,175.699,34.067,156.268
C04292=1070.808,402.401,390.114,175.704,34.075,156.270
C04293=1070.815,402.648,390.072,175.709,34.084,156.272
C04294=1070.824,402.894,390.030,175.715,34.093,156.274
C04295=1070.830,403.140,389.987,175.720,34.101,156.276
C04296=1070.838,403.387,389.946,175.725,34.110,156.278
C04297=1070.845,403.633,389.904,175.730,34.118,156.279
C04298=1070.852,403.879,389.862,175.735,34.128,156.282
C04299=1070.859,404.126,389.821,175.741,34.136,156.284
C04300=1070.867,404.372,389.779,175.746,34.145,156.286
C04301=1070.875,404.619,389.736,175.752,34.154,156.288
C04302=1070.882,404.865,389.694,175.757,34.163,156.290
C04303=1070.890,405.111,389.652,175.762,34.172,156.292
C04304=1070.897,405.357,389.609,175.767,34.181,156.294
C04305=1070.904,405.603,389.567,175.773,34.190,156.296
C04306=1070.912,405.850,389.524,175.778,34.198,156.298
C04307=1070.919,406.096,389.482,175.784,34.208,156.300
C04308=1070.926,406.342,389.440,175.789,34.216,156.302
C04309=1070.934,406.588,389.398,175.795,34.226,156.304
C04310=1070.941,406.835,389.355,175.800,34.235,156.306
C04311=1070.949,407.081,389.313,175.806,34.244,156.308
C04312=1070.956,407.328,389.271,175.810,34.253,156.310
C04313=1070.962,407.574,389.228,175.816,34.262,156.312
C04314=1070.971,407.821,389.186,175.821,34.272,156.315
C04315=1070.978,408.066,389.142,175.827,34.281,156.317
C04316=1070.985,408.312,389.100,175.832,34.290,156.319
C04317=1070.993,408.559,389.058,175.838,34.299,156.321
C04318=1071.000,408.805,389.014,175.844,34.309,156.323
C04319=1071.008,409.052,388.972,175.849,34.318,156.325
C04320=1071.015,409.298,388.930,175.855,34.327,156.327
C04321=1071.022,409.543,388.886,175.860,34.337,156.330
C04322=1071.030,409.790,388.844,175.866,34.346,156.332
C04323=1071.038,410.036,388.801,175.871,34.355,156.334
C04324=1071.045,410.283,388.758,175.877,34.365,156.336
C04325=1071.052,410.528,388.715,175.883,34.374,156.338
C04326=1071.060,410.775,388.672,175.888,34.384,156.341
C04327=1071.068,411.021,388.629,175.894,34.393,156.343
C04328=1071.075,411.267,388.585,175.899,34.403,156.345
C04329=1071.083,411.513,388.543,175.906,34.413,156.347
C04330=1071.091,411.759,388.500,175.912,34.422,156.350
C04331=1071.098,412.005,388.457,175.917,34.432,156.352
C04332=1071.105,412.252,388.414,175.923,34.441,156.354
C04333=1071.114,412.498,388.371,175.928,34.451,156.356
C04334=1071.121,412.744,388.327,175.934,34.461,156.359
C04335=1071.129,412.990,388.284,175.940,34.471,156.361
C04336=1071.137,413.262,388.236,175.946,34.481,156.363
C04337=1071.145,413.534,388.188,175.953,34.492,156.366
C04338=1071.154,413.807,388.141,175.959,34.503,156.368
C04339=1071.163,414.078,388.092,175.966,34.514,156.371
C04340=1071.171,414.324,388.049,175.971,34.524,156.373
C04341=1071.178,414.570,388.005,175.978,34.533,156.376
C04342=1071.186,414.816,387.962,175.984,34.544,156.378
C04343=1071.194,415.062,387.919,175.989,34.553,156.380
C04344=1071.202,415.309,387.875,175.995,34.564,156.383
C04345=1071.209,415.554,387.832,176.001,34.573,156.385
C04346=1071.217,415.801,387.788,176.008,34.584,156.387
C04347=1071.224,416.047,387.743,176.013,34.594,156.390
C04348=1071.232,416.293,387.700,176.019,34.603,156.392
C04349=1071.239,416.539,387.656,176.025,34.614,156.394
C04350=1071.247,416.785,387.612,176.032,34.624,156.397
C04351=1071.255,417.031,387.568,176.037,34.634,156.399
C04352=1071.263,417.277,387.525,176.043,34.644,156.402
C04353=1071.271,417.523,387.480,176.050,34.655,156.404
C04354=1071.279,417.770,387.437,176.056,34.665,156.407
C04355=1071.286,418.015,387.393,176.061,34.676,156.409
C04356=1071.294,418.260,387.349,176.068,34.686,156.412
C04357=1071.302,418.507,387.305,176.074,34.696,156.414
C04358=1071.309,418.753,387.260,176.080,34.707,156.417
C04359=1071.317,418.999,387.216,176.087,34.717,156.419
C04360=1071.325,419.245,387.172,176.092,34.728,156.422
C04361=1071.333,419.491,387.128,176.099,34.738,156.424
C04362=1071.341,419.736,387.083,176.105,34.749,156.427
C04363=1071.349,419.983,387.040,176.111,34.759,156.429
C04364=1071.357,420.228,386.995,176.118,34.769,156.432
C04365=1071.364,420.474,386.950,176.124,34.780,156.434
C04366=1071.372,420.720,386.906,176.130,34.791,156.437
C04367=1071.381,420.966,386.862,176.136,34.802,156.439
C04368=1071.389,421.212,386.817,176.143,34.812,156.442
C04369=1071.396,421.458,386.773,176.149,34.823,156.444
C04370=1071.404,421.703,386.728,176.156,34.834,156.447
C04371=1071.412,421.949,386.684,176.162,34.845,156.450
C04372=1071.420,422.196,386.639,176.169,34.856,156.452
C04373=1071.428,422.442,386.594,176.175,34.867,156.455
C04374=1071.436,422.687,386.549,176.182,34.878,156.457
C04375=1071.444,422.933,386.504,176.187,34.889,156.460
C04376=1071.452,423.179,386.460,176.194,34.899,156.463
C04377=1071.459,423.425,386.415,176.200,34.911,156.465
C04378=1071.468,423.670,386.370,176.207,34.922,156.468
C04379=1071.475,423.917,386.325,176.214,34.933,156.471
C04380=1071.484,424.162,386.280,176.220,34.944,156.474
C04381=1071.491,424.408,386.235,176.227,34.955,156.476
C04382=1071.500,424.653,386.190,176.233,34.966,156.479
C04383=1071.507,424.900,386.144,176.240,34.978,156.482
C04384=1071.516,425.145,386.099,176.247,34.989,156.484
C04385=1071.523,425.391,386.054,176.253,35.000,156.487
C04386=1071.532,425.637,386.009,176.260,35.011,156.490
C04387=1071.540,425.882,385.963,176.267,35.023,156.493
C04388=1071.548,426.128,385.919,176.273,35.034,156.495
C04389=1071.556,426.374,385.873,176.280,35.046,156.498
C04390=1071.565,426.619,385.828,176.287,35.057,156.501
C04391=1071.572,426.865,385.782,176.294,35.068,156.504
C04392=1071.583,427.155,385.729,176.302,35.082,156.507
C04393=1071.592,427.446,385.675,176.310,35.096,156.510
C04394=1071.601,427.737,385.621,176.318,35.110,156.514
C04395=1071.611,428.027,385.567,176.327,35.124,156.517
C04396=1071.619,428.273,385.522,176.334,35.135,156.520
C04397=1071.627,428.519,385.476,176.340,35.147,156.523
C04398=1071.635,428.764,385.430,176.347,35.158,156.526
C04399=1071.644,429.010,385.384,176.354,35.171,156.529
C04400=1071.652,429.255,385.338,176.361,35.182,156.532
C04401=1071.660,429.501,385.292,176.369,35.194,156.535
C04402=1071.668,429.747,385.247,176.376,35.206,156.537
C04403=1071.677,429.992,385.200,176.383,35.218,156.540
C04404=1071.685,430.238,385.154,176.389,35.230,156.543
C04405=1071.693,430.483,385.109,176.396,35.242,156.546
C04406=1071.701,430.729,385.062,176.404,35.254,156.549
C04407=1071.710,430.975,385.016,176.411,35.267,156.552
C04408=1071.718,431.220,384.970,176.418,35.279,156.555
C04409=1071.727,431.466,384.924,176.425,35.291,156.558
C04410=1071.735,431.711,384.878,176.432,35.303,156.561
C04411=1071.743,431.956,384.831,176.440,35.316,156.564
C04412=1071.751,432.202,384.785,176.447,35.328,156.567
C04413=1071.760,432.448,384.738,176.454,35.340,156.571
C04414=1071.768,432.693,384.692,176.462,35.352,156.574
C04415=1071.776,432.938,384.645,176.469,35.365,156.577
C04416=1071.785,433.184,384.599,176.476,35.377,156.580
C04417=1071.793,433.430,384.553,176.484,35.390,156.583
C04418=1071.802,433.675,384.506,176.491,35.403,156.586
C04419=1071.810,433.920,384.460,176.498,35.415,156.589
C04420=1071.817,434.166,384.412,176.506,35.428,156.592
C04421=1071.826,434.411,384.365,176.514,35.440,156.596
C04422=1071.834,434.657,384.319,176.522,35.453,156.599
C04423=1071.843,434.902,384.271,176.529,35.466,156.602
C04424=1071.852,435.147,384.225,176.536,35.479,156.605
C04425=1071.860,435.393,384.178,176.544,35.492,156.608
C04426=1071.869,435.638,384.131,176.551,35.505,156.612
C04427=1071.878,435.883,384.084,176.559,35.518,156.615
C04428=1071.886,436.129,384.037,176.567,35.530,156.618
C04429=1071.895,436.374,383.990,176.575,35.543,156.621
C04430=1071.903,436.619,383.942,176.582,35.556,156.625
C04431=1071.912,436.865,383.895,176.590,35.570,156.628
C04432=1071.920,437.110,383.848,176.598,35.583,156.631
C04433=1071.929,437.355,383.801,176.606,35.596,156.635
C04434=1071.938,437.600,383.754,176.613,35.609,156.638
C04435=1071.946,437.846,383.707,176.622,35.623,156.641
C04436=1071.954,438.091,383.659,176.629,35.636,156.645
C04437=1071.964,438.337,383.611,176.637,35.649,156.648
C04438=1071.972,438.582,383.565,176.646,35.663,156.651
C04439=1071.981,438.827,383.517,176.653,35.676,156.655
C04440=1071.989,439.072,383.469,176.661,35.690,156.658
C04441=1071.998,439.317,383.422,176.669,35.703,156.662
C04442=1072.008,439.563,383.374,176.677,35.717,156.665
C04443=1072.016,439.808,383.326,176.686,35.730,156.669
C04444=1072.025,440.053,383.278,176.694,35.744,156.672
C04445=1072.033,440.298,383.230,176.701,35.758,156.676
C04446=1072.042,440.544,383.182,176.710,35.772,156.679
C04447=1072.051,440.788,383.135,176.718,35.785,156.683
C04448=1072.059,441.018,383.089,176.726,35.798,156.686
C04449=1072.068,441.249,383.044,176.734,35.811,156.689
C04450=1072.075,441.479,382.999,176.742,35.824,156.693
C04451=1072.084,441.710,382.953,176.749,35.838,156.696
C04452=1072.092,441.940,382.909,176.757,35.851,156.699
C04453=1072.100,442.171,382.863,176.765,35.864,156.703
C04454=1072.109,442.401,382.818,176.772,35.878,156.706
C04455=1072.117,442.631,382.773,176.781,35.890,156.710
C04456=1072.127,442.876,382.724,176.789,35.905,156.713
C04457=1072.135,443.121,382.675,176.798,35.919,156.717
C04458=1072.144,443.367,382.627,176.807,35.933,156.721
C04459=1072.153,443.611,382.579,176.815,35.948,156.724
C04460=1072.165,443.936,382.514,176.826,35.967,156.729
C04461=1072.177,444.261,382.450,176.838,35.986,156.734
C04462=1072.189,444.585,382.385,176.849,36.005,156.739
C04463=1072.201,444.910,382.321,176.861,36.025,156.744
C04464=1072.209,445.155,382.272,176.870,36.040,156.748
C04465=1072.218,445.400,382.223,176.878,36.054,156.752
C04466=1072.227,445.645,382.174,176.887,36.069,156.756
C04467=1072.237,445.889,382.125,176.896,36.084,156.760
C04468=1072.246,446.134,382.076,176.905,36.099,156.764
C04469=1072.255,446.380,382.027,176.914,36.114,156.767
C04470=1072.264,446.625,381.978,176.923,36.129,156.772
C04471=1072.274,446.869,381.928,176.933,36.144,156.775
C04472=1072.282,447.114,381.880,176.942,36.159,156.779
C04473=1072.292,447.359,381.830,176.950,36.174,156.783
C04474=1072.301,447.604,381.781,176.959,36.189,156.787
C04475=1072.310,447.848,381.731,176.968,36.204,156.791
C04476=1072.320,448.092,381.682,176.976,36.219,156.795
C04477=1072.329,448.336,381.633,176.985,36.234,156.799
C04478=1072.339,448.580,381.584,176.992,36.249,156.803
C04479=1072.350,448.825,381.536,177.000,36.264,156.807
C04480=1072.362,449.069,381.489,177.007,36.277,156.811
C04481=1072.375,449.315,381.441,177.014,36.291,156.814
C04482=1072.391,449.559,381.396,177.021,36.304,156.818
C04483=1072.406,449.805,381.350,177.028,36.316,156.821
C04484=1072.055,449.804,381.104,177.012,36.461,156.859
C04485=1072.039,449.558,381.149,177.005,36.449,156.856
C04486=1072.024,449.314,381.195,176.998,36.435,156.852
C04487=1072.010,449.069,381.242,176.991,36.422,156.849
C04488=1071.997,448.824,381.289,176.983,36.408,156.845
C04489=1071.986,448.578,381.337,176.976,36.394,156.842
C04490=1071.976,448.334,381.386,176.967,36.379,156.838
C04491=1071.967,448.090,381.435,176.959,36.364,156.834
C04492=1071.957,447.847,381.485,176.951,36.349,156.830
C04493=1071.948,447.602,381.534,176.943,36.334,156.826
C04494=1071.939,447.358,381.584,176.933,36.319,156.822
C04495=1071.930,447.112,381.633,176.924,36.304,156.818
C04496=1071.920,446.869,381.682,176.915,36.288,156.814
C04497=1071.911,446.623,381.731,176.906,36.274,156.810
C04498=1071.902,446.379,381.781,176.896,36.258,156.806
C04499=1071.893,446.133,381.830,176.887,36.243,156.802
C04500=1071.883,445.888,381.878,176.878,36.229,156.798
C04501=1071.875,445.644,381.927,176.869,36.214,156.794
C04502=1071.865,445.399,381.977,176.861,36.199,156.790
C04503=1071.856,445.154,382.026,176.852,36.185,156.786
C04504=1071.847,444.909,382.075,176.842,36.170,156.783
C04505=1071.838,444.664,382.123,176.833,36.155,156.779
C04506=1071.829,444.419,382.173,176.824,36.140,156.775
C04507=1071.820,444.174,382.222,176.816,36.126,156.771
C04508=1071.811,443.929,382.270,176.807,36.112,156.767
C04509=1071.802,443.684,382.318,176.798,36.097,156.764
C04510=1071.793,443.439,382.366,176.790,36.083,156.760
C04511=1071.784,443.194,382.416,176.781,36.068,156.756
C04512=1071.776,442.949,382.464,176.772,36.054,156.753
C04513=1071.766,442.704,382.512,176.764,36.040,156.749
C04514=1071.757,442.459,382.561,176.756,36.026,156.745
C04515=1071.748,442.214,382.609,176.747,36.012,156.742
C04516=1071.740,441.969,382.657,176.739,35.998,156.738
C04517=1071.729,441.691,382.712,176.729,35.982,156.734
C04518=1071.719,441.415,382.767,176.719,35.966,156.730
C04519=1071.709,441.138,382.821,176.710,35.950,156.726
C04520=1071.700,440.861,382.876,176.700,35.935,156.722
C04521=1071.691,440.616,382.923,176.692,35.921,156.718
C04522=1071.681,440.370,382.971,176.684,35.907,156.715
C04523=1071.673,440.125,383.019,176.676,35.893,156.711
C04524=1071.664,439.881,383.067,176.667,35.880,156.708
C04525=1071.655,439.635,383.115,176.659,35.866,156.704
C04526=1071.646,439.390,383.163,176.652,35.852,156.701
C04527=1071.638,439.145,383.210,176.643,35.839,156.697
C04528=1071.629,438.900,383.258,176.635,35.825,156.694
C04529=1071.621,438.655,383.306,176.626,35.812,156.690
C04530=1071.611,438.409,383.353,176.619,35.798,156.687
C04531=1071.603,438.164,383.401,176.611,35.785,156.684
C04532=1071.595,437.919,383.448,176.602,35.772,156.680
C04533=1071.586,437.674,383.496,176.595,35.759,156.677
C04534=1071.577,437.428,383.543,176.587,35.745,156.673
C04535=1071.568,437.183,383.590,176.579,35.732,156.670
C04536=1071.559,436.937,383.637,176.571,35.719,156.667
C04537=1071.551,436.692,383.685,176.563,35.706,156.664
C04538=1071.542,436.446,383.732,176.556,35.693,156.660
C04539=1071.534,436.202,383.779,176.547,35.680,156.657
C04540=1071.525,435.956,383.826,176.540,35.667,156.654
C04541=1071.517,435.733,383.869,176.532,35.655,156.651
C04542=1071.509,435.511,383.912,176.526,35.644,156.648
C04543=1071.501,435.288,383.955,176.519,35.632,156.645
C04544=1071.494,435.065,383.997,176.512,35.620,156.642
C04545=1071.486,434.842,384.040,176.505,35.609,156.639
C04546=1071.478,434.619,384.083,176.497,35.597,156.636
C04547=1071.470,434.396,384.125,176.491,35.586,156.633
C04548=1071.462,434.173,384.168,176.484,35.574,156.630
C04549=1071.454,433.928,384.214,176.476,35.562,156.627
C04550=1071.446,433.683,384.261,176.469,35.549,156.624
C04551=1071.437,433.437,384.308,176.462,35.537,156.621
C04552=1071.429,433.192,384.354,176.454,35.524,156.618
C04553=1071.421,432.946,384.402,176.447,35.511,156.615
C04554=1071.413,432.700,384.448,176.439,35.499,156.611
C04555=1071.405,432.455,384.494,176.432,35.487,156.608
C04556=1071.396,432.209,384.541,176.425,35.474,156.605
C04557=1071.388,431.964,384.588,176.417,35.462,156.602
C04558=1071.380,431.719,384.634,176.410,35.449,156.599
C04559=1071.372,431.473,384.680,176.402,35.437,156.596
C04560=1071.362,431.228,384.726,176.395,35.425,156.593
C04561=1071.354,430.982,384.772,176.388,35.413,156.590
C04562=1071.346,430.737,384.819,176.381,35.401,156.587
C04563=1071.338,430.491,384.865,176.373,35.389,156.584
C04564=1071.329,430.245,384.911,176.366,35.377,156.581
C04565=1071.321,430.000,384.956,176.359,35.365,156.578
C04566=1071.312,429.754,385.003,176.351,35.353,156.575
C04567=1071.304,429.508,385.049,176.345,35.341,156.572
C04568=1071.296,429.263,385.095,176.338,35.329,156.569
C04569=1071.288,429.017,385.141,176.331,35.317,156.566
C04570=1071.280,428.772,385.186,176.323,35.305,156.563
C04571=1071.271,428.526,385.232,176.316,35.294,156.561
C04572=1071.264,428.281,385.278,176.309,35.282,156.558
C04573=1071.252,427.944,385.341,176.299,35.266,156.554
C04574=1071.241,427.606,385.404,176.291,35.250,156.550
C04575=1071.230,427.269,385.466,176.281,35.234,156.546
C04576=1071.219,426.932,385.529,176.272,35.218,156.542
C04577=1071.210,426.686,385.575,176.265,35.206,156.539
C04578=1071.202,426.440,385.620,176.257,35.195,156.536
C04579=1071.193,426.194,385.665,176.250,35.183,156.534
C04580=1071.186,425.949,385.711,176.244,35.172,156.531
C04581=1071.177,425.704,385.756,176.237,35.161,156.528
C04582=1071.170,425.457,385.801,176.230,35.150,156.525
C04583=1071.161,425.212,385.846,176.224,35.138,156.522
C04584=1071.154,424.966,385.892,176.217,35.127,156.520
C04585=1071.145,424.720,385.936,176.210,35.116,156.517
C04586=1071.137,424.474,385.982,176.204,35.105,156.514
C04587=1071.129,424.229,386.026,176.197,35.094,156.512
C04588=1071.121,423.983,386.072,176.191,35.083,156.509
C04589=1071.113,423.737,386.117,176.184,35.071,156.506
C04590=1071.104,423.492,386.162,176.177,35.060,156.504
C04591=1071.097,423.246,386.207,176.171,35.049,156.501
C04592=1071.089,423.001,386.252,176.164,35.038,156.498
C04593=1071.081,422.754,386.297,176.158,35.027,156.496
C04594=1071.073,422.508,386.341,176.151,35.016,156.493
C04595=1071.065,422.262,386.386,176.145,35.005,156.490
C04596=1071.057,422.017,386.431,176.138,34.995,156.488
C04597=1071.049,421.771,386.476,176.132,34.983,156.485
C04598=1071.042,421.525,386.521,176.125,34.973,156.482
C04599=1071.034,421.279,386.565,176.119,34.962,156.480
C04600=1071.025,421.034,386.609,176.112,34.951,156.477
C04601=1071.018,420.787,386.655,176.106,34.941,156.475
C04602=1071.009,420.541,386.699,176.099,34.930,156.472
C04603=1071.001,420.295,386.743,176.093,34.919,156.470
C04604=1070.993,420.050,386.788,176.086,34.909,156.467
C04605=1070.985,419.804,386.832,176.080,34.898,156.465
C04606=1070.978,419.557,386.876,176.074,34.888,156.462
C04607=1070.970,419.311,386.920,176.067,34.877,156.459
C04608=1070.962,419.066,386.965,176.062,34.867,156.457
C04609=1070.954,418.820,387.009,176.055,34.856,156.454
C04610=1070.946,418.574,387.053,176.049,34.846,156.452
C04611=1070.938,418.328,387.097,176.043,34.836,156.449
C04612=1070.930,418.082,387.141,176.036,34.825,156.447
C04613=1070.922,417.836,387.185,176.030,34.815,156.445
C04614=1070.915,417.591,387.229,176.025,34.805,156.442
C04615=1070.908,417.344,387.273,176.018,34.794,156.440
C04616=1070.900,417.098,387.318,176.012,34.784,156.437
C04617=1070.892,416.852,387.361,176.006,34.774,156.435
C04618=1070.884,416.606,387.406,175.999,34.764,156.432
C04619=1070.876,416.360,387.449,175.993,34.753,156.430
C04620=1070.869,416.115,387.493,175.988,34.743,156.428
C04621=1070.861,415.868,387.537,175.982,34.733,156.425
C04622=1070.853,415.622,387.580,175.975,34.723,156.423
C04623=1070.845,415.376,387.624,175.969,34.713,156.420
C04624=1070.838,415.131,387.668,175.964,34.703,156.418
C04625=1070.830,414.884,387.712,175.958,34.693,156.416
C04626=1070.822,414.638,387.755,175.951,34.683,156.413
C04627=1070.815,414.391,387.799,175.945,34.673,156.411
C04628=1070.807,414.145,387.842,175.940,34.663,156.409
C04629=1070.798,413.872,387.890,175.933,34.653,156.406
C04630=1070.789,413.598,387.939,175.927,34.642,156.404
C04631=1070.781,413.324,387.987,175.920,34.631,156.401
C04632=1070.772,413.051,388.035,175.913,34.620,156.398
C04633=1070.764,412.805,388.078,175.908,34.610,156.396
C04634=1070.757,412.559,388.122,175.902,34.601,156.394
C04635=1070.750,412.312,388.165,175.896,34.591,156.392
C04636=1070.741,412.066,388.208,175.891,34.581,156.389
C04637=1070.734,411.821,388.251,175.884,34.571,156.387
C04638=1070.726,411.574,388.295,175.878,34.562,156.385
C04639=1070.719,411.328,388.337,175.873,34.552,156.383
C04640=1070.711,411.082,388.380,175.867,34.543,156.380
C04641=1070.703,410.835,388.424,175.861,34.533,156.378
C04642=1070.696,410.589,388.466,175.856,34.524,156.376
C04643=1070.688,410.343,388.509,175.850,34.514,156.374
C04644=1070.681,410.097,388.553,175.844,34.505,156.372
C04645=1070.674,409.851,388.595,175.839,34.495,156.369
C04646=1070.665,409.605,388.638,175.833,34.486,156.367
C04647=1070.658,409.359,388.681,175.827,34.477,156.365
C04648=1070.651,409.112,388.724,175.822,34.468,156.363
C04649=1070.643,408.866,388.766,175.816,34.458,156.361
C04650=1070.636,408.619,388.809,175.811,34.449,156.359
C04651=1070.628,408.374,388.852,175.805,34.439,156.356
C04652=1070.621,408.128,388.894,175.799,34.431,156.354
C04653=1070.613,407.881,388.937,175.794,34.421,156.352
C04654=1070.606,407.635,388.980,175.788,34.412,156.350
C04655=1070.599,407.389,389.022,175.783,34.403,156.348
C04656=1070.591,407.142,389.065,175.777,34.394,156.346
C04657=1070.584,406.896,389.108,175.771,34.384,156.343
C04658=1070.577,406.650,389.150,175.767,34.376,156.341
C04659=1070.569,406.404,389.193,175.761,34.366,156.339
C04660=1070.561,406.158,389.235,175.756,34.357,156.337
C04661=1070.554,405.911,389.278,175.750,34.348,156.335
C04662=1070.547,405.665,389.320,175.745,34.340,156.333
C04663=1070.539,405.419,389.362,175.739,34.330,156.331
C04664=1070.532,405.172,389.405,175.734,34.321,156.329
C04665=1070.524,404.926,389.447,175.728,34.312,156.327
C04666=1070.518,404.680,389.488,175.724,34.303,156.325
C04667=1070.510,404.434,389.530,175.718,34.295,156.323
C04668=1070.503,404.187,389.573,175.712,34.286,156.321
C04669=1070.495,403.941,389.615,175.707,34.277,156.319
C04670=1070.487,403.695,389.657,175.701,34.268,156.317
C04671=1070.481,403.448,389.699,175.696,34.260,156.315
C04672=1070.473,403.202,389.741,175.691,34.251,156.313
C04673=1070.466,402.956,389.783,175.686,34.242,156.311
C04674=1070.458,402.709,389.825,175.680,34.233,156.309
C04675=1070.451,402.462,389.867,175.675,34.224,156.307
C04676=1070.443,402.216,389.909,175.671,34.216,156.305
C04677=1070.436,401.970,389.950,175.665,34.207,156.303
C04678=1070.428,401.724,389.992,175.660,34.199,156.301
C04679=1070.421,401.477,390.033,175.654,34.190,156.299
C04680=1070.414,401.231,390.076,175.650,34.182,156.297
C04681=1070.407,400.984,390.117,175.644,34.173,156.295
C04682=1070.399,400.738,390.159,175.639,34.165,156.293
C04683=1070.392,400.492,390.200,175.633,34.156,156.291
C04684=1070.385,400.246,390.242,175.629,34.148,156.289
C04685=1070.377,399.975,390.288,175.623,34.139,156.287
C04686=1070.369,399.706,390.333,175.617,34.129,156.285
C04687=1070.361,399.435,390.378,175.611,34.120,156.283
C04688=1070.353,399.166,390.424,175.606,34.111,156.281
C04689=1070.346,398.919,390.465,175.601,34.103,156.279
C04690=1070.339,398.673,390.506,175.596,34.094,156.277
C04691=1070.331,398.427,390.548,175.591,34.086,156.275
C04692=1070.324,398.180,390.590,175.585,34.077,156.273
C04693=1070.317,397.933,390.631,175.581,34.069,156.271
C04694=1070.309,397.687,390.672,175.575,34.061,156.270
C04695=1070.303,397.441,390.713,175.571,34.053,156.268
C04696=1070.295,397.194,390.754,175.566,34.045,156.266
C04697=1070.288,396.948,390.795,175.560,34.037,156.264
C04698=1070.281,396.701,390.837,175.556,34.028,156.262
C04699=1070.273,396.454,390.878,175.551,34.020,156.260
C04700=1070.266,396.208,390.919,175.545,34.012,156.259
C04701=1070.259,395.962,390.960,175.541,34.004,156.257
C04702=1070.251,395.716,391.001,175.535,33.996,156.255
C04703=1070.244,395.469,391.042,175.531,33.988,156.253
C04704=1070.237,395.222,391.082,175.526,33.980,156.251
C04705=1070.231,394.976,391.123,175.520,33.972,156.250
C04706=1070.223,394.729,391.164,175.516,33.964,156.248
C04707=1070.216,394.483,391.206,175.511,33.956,156.246
C04708=1070.209,394.237,391.247,175.506,33.948,156.244
C04709=1070.202,393.990,391.287,175.501,33.940,156.242
C04710=1070.194,393.743,391.328,175.497,33.932,156.241
C04711=1070.188,393.498,391.369,175.491,33.924,156.239
C04712=1070.181,393.250,391.409,175.487,33.917,156.237
C04713=1070.173,393.004,391.450,175.481,33.908,156.235
C04714=1070.166,392.758,391.490,175.477,33.901,156.234
C04715=1070.159,392.511,391.531,175.472,33.893,156.232
C04716=1070.152,392.264,391.571,175.467,33.885,156.230
C04717=1070.144,392.018,391.612,175.462,33.877,156.228
C04718=1070.137,391.771,391.652,175.457,33.869,156.227
C04719=1070.131,391.525,391.693,175.453,33.862,156.225
C04720=1070.123,391.278,391.733,175.447,33.854,156.223
C04721=1070.116,391.032,391.774,175.443,33.846,156.222
C04722=1070.109,390.785,391.815,175.438,33.839,156.220
C04723=1070.102,390.539,391.854,175.433,33.831,156.218
C04724=1070.095,390.292,391.895,175.428,33.824,156.217
C04725=1070.088,390.046,391.935,175.424,33.816,156.215
C04726=1070.081,389.799,391.975,175.418,33.808,156.213
C04727=1070.074,389.553,392.015,175.414,33.801,156.211
C04728=1070.066,389.306,392.056,175.410,33.793,156.210
C04729=1070.059,389.060,392.096,175.405,33.786,156.208
C04730=1070.052,388.813,392.136,175.400,33.778,156.207
C04731=1070.045,388.566,392.176,175.395,33.771,156.205
C04732=1070.038,388.319,392.216,175.391,33.763,156.203
C04733=1070.031,388.073,392.256,175.386,33.756,156.202
C04734=1070.023,387.826,392.296,175.381,33.749,156.200
C04735=1070.016,387.580,392.335,175.376,33.741,156.198
C04736=1070.010,387.333,392.375,175.372,33.733,156.197
C04737=1070.002,387.086,392.415,175.367,33.726,156.195
C04738=1069.996,386.840,392.456,175.362,33.719,156.193
C04739=1069.989,386.594,392.495,175.358,33.712,156.192
C04740=1069.981,386.347,392.535,175.353,33.704,156.190
C04741=1069.974,386.093,392.576,175.348,33.696,156.189
C04742=1069.967,385.839,392.617,175.343,33.689,156.187
C04743=1069.960,385.585,392.658,175.339,33.681,156.185
C04744=1069.953,385.330,392.699,175.334,33.674,156.184
C04745=1069.946,385.084,392.739,175.329,33.667,156.182
C04746=1069.939,384.837,392.778,175.325,33.659,156.180
C04747=1069.933,384.590,392.818,175.320,33.652,156.179
C04748=1069.925,384.344,392.857,175.316,33.645,156.177
C04749=1069.918,384.097,392.897,175.312,33.638,156.176
C04750=1069.912,383.850,392.937,175.306,33.631,156.174
C04751=1069.904,383.604,392.976,175.302,33.623,156.173
C04752=1069.897,383.358,393.016,175.298,33.616,156.171
C04753=1069.891,383.110,393.056,175.293,33.609,156.169
C04754=1069.884,382.864,393.095,175.289,33.602,156.168
C04755=1069.877,382.617,393.134,175.284,33.595,156.166
C04756=1069.870,382.370,393.174,175.280,33.588,156.165
C04757=1069.864,382.123,393.213,175.275,33.580,156.163
C04758=1069.856,381.877,393.253,175.271,33.574,156.162
C04759=1069.850,381.630,393.291,175.266,33.566,156.160
C04760=1069.843,381.384,393.332,175.261,33.559,156.159
C04761=1069.836,381.136,393.371,175.257,33.552,156.157
C04762=1069.829,380.890,393.410,175.253,33.545,156.156
C04763=1069.822,380.643,393.449,175.249,33.539,156.154
C04764=1069.815,380.396,393.488,175.244,33.532,156.153
C04765=1069.808,380.150,393.527,175.239,33.524,156.151
C04766=1069.801,379.903,393.566,175.235,33.518,156.150
C04767=1069.795,379.656,393.604,175.231,33.511,156.148
C04768=1069.787,379.409,393.644,175.226,33.504,156.147
C04769=1069.780,379.162,393.683,175.222,33.497,156.145
C04770=1069.773,378.915,393.722,175.217,33.490,156.144
C04771=1069.767,378.669,393.761,175.213,33.484,156.142
C04772=1069.760,378.422,393.800,175.208,33.477,156.141
C04773=1069.753,378.175,393.839,175.204,33.470,156.139
C04774=1069.746,377.928,393.877,175.200,33.463,156.138
C04775=1069.739,377.681,393.916,175.196,33.456,156.136
C04776=1069.732,377.435,393.955,175.190,33.449,156.135
C04777=1069.726,377.188,393.994,175.186,33.443,156.134
C04778=1069.719,376.941,394.033,175.182,33.436,156.132
C04779=1069.712,376.694,394.072,175.178,33.429,156.131
C04780=1069.705,376.447,394.110,175.174,33.422,156.129
C04781=1069.698,376.200,394.149,175.170,33.416,156.128
C04782=1069.691,375.954,394.188,175.165,33.409,156.126
C04783=1069.684,375.707,394.226,175.160,33.402,156.125
C04784=1069.678,375.460,394.264,175.156,33.396,156.123
C04785=1069.671,375.213,394.303,175.152,33.389,156.122
C04786=1069.665,374.967,394.342,175.148,33.382,156.121
C04787=1069.658,374.720,394.381,175.144,33.376,156.119
C04788=1069.651,374.472,394.419,175.139,33.369,156.118
C04789=1069.644,374.226,394.458,175.135,33.362,156.116
C04790=1069.638,373.979,394.496,175.131,33.356,156.115
C04791=1069.631,373.732,394.535,175.126,33.349,156.114
C04792=1069.625,373.485,394.573,175.122,33.343,156.112
C04793=1069.618,373.250,394.610,175.118,33.337,156.111
C04794=1069.611,373.014,394.646,175.114,33.330,156.110
C04795=1069.605,372.778,394.683,175.110,33.324,156.108
C04796=1069.599,372.543,394.719,175.106,33.318,156.107
C04797=1069.592,372.308,394.756,175.102,33.312,156.106
C04798=1069.585,372.072,394.792,175.098,33.306,156.104
C04799=1069.579,371.836,394.829,175.093,33.300,156.103
C04800=1069.572,371.601,394.865,175.090,33.293,156.102
C04801=1069.566,371.354,394.903,175.085,33.287,156.100
C04802=1069.559,371.107,394.941,175.081,33.281,156.099
C04803=1069.552,370.860,394.980,175.077,33.274,156.098
C04804=1069.545,370.613,395.017,175.073,33.268,156.096
C04805=1069.538,370.366,395.055,175.069,33.262,156.095
C04806=1069.532,370.120,395.093,175.065,33.255,156.094
C04807=1069.525,369.872,395.131,175.061,33.249,156.092
C04808=1069.518,369.625,395.169,175.057,33.242,156.091
C04809=1069.512,369.378,395.207,175.052,33.236,156.090
C04810=1069.505,369.132,395.245,175.048,33.230,156.088
C04811=1069.498,368.884,395.283,175.044,33.224,156.087
C04812=1069.491,368.637,395.321,175.040,33.218,156.086
C04813=1069.485,368.391,395.358,175.036,33.211,156.084
C04814=1069.478,368.143,395.396,175.032,33.205,156.083
C04815=1069.472,367.896,395.434,175.028,33.199,156.082
C04816=1069.465,367.649,395.472,175.024,33.192,156.080
C04817=1069.458,367.402,395.510,175.020,33.186,156.079
C04818=1069.451,367.155,395.547,175.015,33.180,156.078
C04819=1069.445,366.908,395.585,175.011,33.174,156.077
C04820=1069.438,366.661,395.622,175.007,33.167,156.075
C04821=1069.432,366.414,395.660,175.003,33.161,156.074
C04822=1069.425,366.167,395.698,174.998,33.155,156.073
C04823=1069.419,365.920,395.736,174.994,33.149,156.071
C04824=1069.412,365.673,395.773,174.991,33.143,156.070
C04825=1069.405,365.426,395.811,174.987,33.136,156.069
C04826=1069.399,365.179,395.848,174.983,33.131,156.068
C04827=1069.392,364.932,395.886,174.979,33.124,156.066
C04828=1069.386,364.685,395.924,174.975,33.118,156.065
C04829=1069.379,364.437,395.961,174.971,33.112,156.064
C04830=1069.373,364.191,395.998,174.967,33.106,156.062
C04831=1069.365,363.944,396.036,174.963,33.100,156.061
C04832=1069.360,363.697,396.073,174.959,33.094,156.060
C04833=1069.353,363.449,396.110,174.955,33.088,156.059
C04834=1069.345,363.202,396.148,174.951,33.082,156.057
C04835=1069.339,362.955,396.184,174.947,33.076,156.056
C04836=1069.332,362.707,396.222,174.943,33.070,156.055
C04837=1069.326,362.461,396.260,174.939,33.064,156.054
C04838=1069.319,362.213,396.296,174.935,33.058,156.053
C04839=1069.312,361.967,396.334,174.931,33.052,156.051
C04840=1069.306,361.719,396.371,174.926,33.046,156.050
C04841=1069.299,361.472,396.408,174.922,33.040,156.049
C04842=1069.293,361.225,396.445,174.918,33.035,156.048
C04843=1069.286,360.978,396.482,174.914,33.029,156.046
C04844=1069.280,360.731,396.518,174.910,33.022,156.045
C04845=1069.273,360.484,396.557,174.907,33.017,156.044
C04846=1069.267,360.237,396.593,174.903,33.011,156.043
C04847=1069.259,359.989,396.631,174.899,33.005,156.041
C04848=1069.253,359.742,396.667,174.895,32.999,156.040
C04849=1069.247,359.515,396.702,174.891,32.994,156.039
C04850=1069.241,359.288,396.735,174.888,32.988,156.038
C04851=1069.235,359.061,396.769,174.884,32.983,156.037
C04852=1069.229,358.835,396.803,174.881,32.978,156.036
C04853=1069.223,358.607,396.836,174.877,32.972,156.035
C04854=1069.217,358.381,396.870,174.873,32.967,156.034
C04855=1069.211,358.153,396.903,174.870,32.962,156.033
C04856=1069.205,357.926,396.938,174.866,32.957,156.032
C04857=1069.199,357.679,396.974,174.862,32.951,156.030
C04858=1069.192,357.432,397.011,174.859,32.945,156.029
C04859=1069.185,357.184,397.048,174.855,32.939,156.028
C04860=1069.179,356.938,397.085,174.851,32.933,156.027
C04861=1069.172,356.691,397.121,174.847,32.928,156.026
C04862=1069.165,356.443,397.158,174.843,32.922,156.025
C04863=1069.159,356.196,397.195,174.839,32.916,156.023
C04864=1069.153,355.949,397.231,174.835,32.911,156.022
C04865=1069.146,355.702,397.267,174.832,32.905,156.021
C04866=1069.139,355.454,397.304,174.828,32.900,156.020
C04867=1069.132,355.207,397.340,174.824,32.894,156.019
C04868=1069.126,354.960,397.377,174.820,32.888,156.017
C04869=1069.120,354.713,397.413,174.816,32.883,156.016
C04870=1069.113,354.466,397.450,174.812,32.877,156.015
C04871=1069.106,354.218,397.486,174.809,32.871,156.014
C04872=1069.100,353.971,397.522,174.805,32.866,156.013
C04873=1069.094,353.724,397.558,174.801,32.860,156.012
C04874=1069.088,353.477,397.595,174.797,32.854,156.011
C04875=1069.081,353.229,397.632,174.793,32.849,156.010
C04876=1069.074,352.982,397.668,174.790,32.843,156.008
C04877=1069.068,352.735,397.705,174.786,32.838,156.007
C04878=1069.062,352.487,397.740,174.782,32.832,156.006
C04879=1069.055,352.240,397.776,174.778,32.826,156.005
C04880=1069.049,351.993,397.813,174.775,32.821,156.004
C04881=1069.042,351.745,397.849,174.771,32.815,156.003
C04882=1069.036,351.498,397.885,174.767,32.810,156.002
C04883=1069.029,351.251,397.922,174.763,32.804,156.001
C04884=1069.023,351.003,397.957,174.759,32.799,155.999
C04885=1069.016,350.756,397.993,174.756,32.794,155.998
C04886=1069.010,350.509,398.029,174.752,32.788,155.997
C04887=1069.002,350.261,398.065,174.748,32.782,155.996
C04888=1068.996,350.014,398.102,174.744,32.777,155.995
C04889=1068.990,349.767,398.137,174.741,32.772,155.994
C04890=1068.983,349.520,398.173,174.737,32.766,155.993
C04891=1068.977,349.272,398.209,174.733,32.761,155.992
C04892=1068.971,349.025,398.245,174.729,32.755,155.991
C04893=1068.964,348.778,398.280,174.726,32.750,155.990
C04894=1068.958,348.530,398.316,174.722,32.745,155.989
C04895=1068.952,348.283,398.353,174.718,32.739,155.987
C04896=1068.945,348.036,398.388,174.715,32.734,155.986
C04897=1068.938,347.789,398.424,174.711,32.728,155.985
C04898=1068.932,347.541,398.460,174.707,32.723,155.984
C04899=1068.926,347.294,398.495,174.703,32.718,155.983
C04900=1068.919,347.047,398.532,174.701,32.712,155.982
C04901=1068.913,346.799,398.567,174.697,32.707,155.981
C04902=1068.906,346.551,398.602,174.693,32.702,155.980
C04903=1068.900,346.304,398.638,174.690,32.696,155.979
C04904=1068.893,346.057,398.674,174.686,32.691,155.978
C04905=1068.888,345.831,398.706,174.683,32.686,155.977
C04906=1068.882,345.607,398.738,174.679,32.681,155.976
C04907=1068.876,345.382,398.771,174.676,32.676,155.975
C04908=1068.870,345.156,398.803,174.673,32.672,155.974
C04909=1068.864,344.931,398.835,174.669,32.667,155.973
C04910=1068.858,344.706,398.868,174.666,32.662,155.972
C04911=1068.853,344.481,398.900,174.663,32.657,155.971
C04912=1068.847,344.256,398.933,174.659,32.652,155.970
C04913=1068.841,344.009,398.968,174.656,32.647,155.969
C04914=1068.834,343.761,399.003,174.652,32.642,155.968
C04915=1068.828,343.514,399.039,174.648,32.637,155.967
C04916=1068.822,343.266,399.074,174.645,32.631,155.966
C04917=1068.815,343.019,399.109,174.641,32.626,155.965
C04918=1068.809,342.771,399.145,174.637,32.621,155.964
C04919=1068.802,342.524,399.180,174.634,32.616,155.963
C04920=1068.795,342.276,399.215,174.630,32.611,155.962
C04921=1068.789,342.029,399.251,174.626,32.605,155.961
C04922=1068.782,341.781,399.286,174.623,32.601,155.960
C04923=1068.776,341.533,399.320,174.620,32.595,155.959
C04924=1068.771,341.286,399.356,174.616,32.590,155.958
C04925=1068.764,341.039,399.391,174.613,32.585,155.957
C04926=1068.757,340.792,399.426,174.609,32.580,155.956
C04927=1068.750,340.544,399.461,174.606,32.574,155.955
C04928=1068.744,340.297,399.497,174.602,32.570,155.954
C04929=1068.738,340.049,399.531,174.598,32.564,155.953
C04930=1068.732,339.802,399.566,174.595,32.559,155.952
C04931=1068.726,339.554,399.602,174.591,32.554,155.951
C04932=1068.719,339.306,399.636,174.588,32.549,155.950
C04933=1068.712,339.059,399.671,174.584,32.544,155.949
C04934=1068.706,338.812,399.706,174.580,32.539,155.948
C04935=1068.700,338.564,399.741,174.577,32.533,155.946
C04936=1068.694,338.317,399.776,174.573,32.529,155.946
C04937=1068.687,338.069,399.811,174.570,32.523,155.944
C04938=1068.681,337.822,399.845,174.567,32.518,155.944
C04939=1068.675,337.574,399.881,174.564,32.513,155.942
C04940=1068.669,337.326,399.916,174.560,32.508,155.942
C04941=1068.662,337.080,399.950,174.556,32.503,155.941
C04942=1068.656,336.832,399.985,174.553,32.498,155.940
C04943=1068.649,336.584,400.020,174.549,32.493,155.939
C04944=1068.643,336.336,400.054,174.546,32.488,155.938
C04945=1068.637,336.090,400.089,174.542,32.483,155.937
C04946=1068.630,335.842,400.123,174.539,32.479,155.936
C04947=1068.623,335.594,400.159,174.535,32.473,155.935
C04948=1068.617,335.347,400.193,174.532,32.468,155.934
C04949=1068.611,335.099,400.227,174.528,32.464,155.933
C04950=1068.604,334.852,400.262,174.524,32.458,155.932
C04951=1068.598,334.604,400.296,174.522,32.453,155.931
C04952=1068.592,334.357,400.331,174.518,32.449,155.930
C04953=1068.585,334.109,400.366,174.515,32.444,155.929
C04954=1068.579,333.862,400.400,174.511,32.438,155.928
C04955=1068.573,333.614,400.434,174.508,32.434,155.927
C04956=1068.566,333.366,400.469,174.504,32.429,155.926
C04957=1068.560,333.119,400.503,174.501,32.424,155.925
C04958=1068.554,332.871,400.538,174.497,32.419,155.924
C04959=1068.548,332.624,400.572,174.494,32.414,155.923
C04960=1068.541,332.376,400.606,174.490,32.409,155.922
C04961=1068.536,332.148,400.639,174.487,32.404,155.921
C04962=1068.530,331.921,400.670,174.484,32.400,155.920
C04963=1068.524,331.694,400.701,174.482,32.395,155.919
C04964=1068.519,331.466,400.733,174.479,32.391,155.919
C04965=1068.513,331.238,400.764,174.475,32.386,155.918
C04966=1068.506,331.011,400.796,174.472,32.382,155.917
C04967=1068.501,330.783,400.828,174.469,32.378,155.916
C04968=1068.495,330.555,400.859,174.466,32.373,155.915
C04969=1068.488,330.307,400.892,174.462,32.368,155.914
C04970=1068.482,330.060,400.926,174.459,32.364,155.913
C04971=1068.476,329.812,400.961,174.455,32.359,155.913
C04972=1068.469,329.565,400.994,174.452,32.355,155.912
C04973=1068.463,329.317,401.029,174.449,32.350,155.911
C04974=1068.457,329.070,401.063,174.446,32.345,155.910
C04975=1068.450,328.822,401.097,174.442,32.340,155.909
C04976=1068.444,328.575,401.131,174.439,32.335,155.908
C04977=1068.437,328.327,401.165,174.435,32.330,155.907
C04978=1068.430,328.079,401.199,174.432,32.326,155.906
C04979=1068.425,327.831,401.232,174.429,32.321,155.905
C04980=1068.418,327.584,401.266,174.425,32.317,155.904
C04981=1068.412,327.336,401.300,174.422,32.312,155.903
C04982=1068.405,327.089,401.334,174.418,32.307,155.902
C04983=1068.399,326.841,401.368,174.416,32.302,155.901
C04984=1068.393,326.594,401.401,174.412,32.297,155.901
C04985=1068.386,326.346,401.435,174.409,32.293,155.900
C04986=1068.380,326.099,401.469,174.405,32.288,155.899
C04987=1068.373,325.850,401.502,174.402,32.283,155.898
C04988=1068.367,325.603,401.536,174.399,32.279,155.897
C04989=1068.360,325.355,401.570,174.395,32.274,155.896
C04990=1068.355,325.107,401.604,174.392,32.270,155.895
C04991=1068.349,324.860,401.638,174.388,32.265,155.894
C04992=1068.341,324.613,401.671,174.386,32.260,155.893
C04993=1068.336,324.365,401.705,174.383,32.256,155.893
C04994=1068.329,324.117,401.739,174.379,32.251,155.892
C04995=1068.323,323.869,401.772,174.376,32.246,155.891
C04996=1068.317,323.622,401.805,174.372,32.241,155.890
C04997=1068.310,323.373,401.839,174.369,32.237,155.889
C04998=1068.304,323.126,401.873,174.366,32.232,155.888
C04999=1068.298,322.879,401.906,174.362,32.227,155.887
C05000=1068.291,322.631,401.940,174.359,32.222,155.886
C05001=1068.285,322.383,401.973,174.357,32.218,155.885
C05002=1068.279,322.136,402.007,174.353,32.213,155.884
C05003=1068.273,321.888,402.040,174.350,32.209,155.884
C05004=1068.266,321.640,402.074,174.346,32.204,155.883
C05005=1068.261,321.393,402.107,174.343,32.199,155.882
C05006=1068.254,321.145,402.140,174.340,32.195,155.881
C05007=1068.248,320.898,402.174,174.336,32.190,155.880
C05008=1068.242,320.649,402.207,174.333,32.186,155.879
C05009=1068.236,320.401,402.240,174.331,32.181,155.878
C05010=1068.229,320.154,402.274,174.327,32.176,155.877
C05011=1068.224,319.907,402.307,174.324,32.172,155.877
C05012=1068.218,319.659,402.340,174.321,32.167,155.876
C05013=1068.211,319.411,402.374,174.317,32.162,155.875
C05014=1068.205,319.163,402.407,174.314,32.158,155.874
C05015=1068.199,318.916,402.440,174.311,32.153,155.873
C05016=1068.193,318.668,402.473,174.307,32.149,155.872
C05017=1068.187,318.438,402.505,174.305,32.144,155.871
C05018=1068.181,318.207,402.535,174.302,32.140,155.871
C05019=1068.175,317.976,402.566,174.299,32.136,155.870
C05020=1068.170,317.745,402.597,174.296,32.132,155.869
C05021=1068.164,317.515,402.628,174.293,32.127,155.868
C05022=1068.159,317.284,402.658,174.290,32.123,155.867
C05023=1068.153,317.054,402.689,174.287,32.119,155.866
C05024=1068.148,316.823,402.720,174.284,32.115,155.866
C05025=1068.141,316.575,402.753,174.282,32.110,155.865
C05026=1068.135,316.328,402.787,174.278,32.105,155.864
C05027=1068.129,316.080,402.820,174.275,32.101,155.863
C05028=1068.123,315.833,402.852,174.272,32.096,155.862
C05029=1068.117,315.585,402.886,174.268,32.092,155.861
C05030=1068.111,315.337,402.918,174.265,32.087,155.860
C05031=1068.105,315.089,402.952,174.262,32.082,155.860
C05032=1068.099,314.842,402.985,174.260,32.078,155.859
C05033=1068.093,314.594,403.017,174.256,32.073,155.858
C05034=1068.087,314.346,403.051,174.253,32.069,155.857
C05035=1068.081,314.098,403.083,174.250,32.064,155.856
C05036=1068.074,313.850,403.116,174.246,32.060,155.855
C05037=1068.068,313.602,403.149,174.243,32.055,155.854
C05038=1068.062,313.355,403.181,174.240,32.051,155.854
C05039=1068.055,313.107,403.214,174.238,32.047,155.853
C05040=1068.049,312.859,403.247,174.234,32.042,155.852
C05041=1068.043,312.611,403.279,174.231,32.038,155.851
C05042=1068.036,312.364,403.311,174.228,32.034,155.850
C05043=1068.030,312.116,403.344,174.225,32.029,155.849
C05044=1068.024,311.869,403.376,174.221,32.024,155.849
C05045=1068.018,311.621,403.408,174.218,32.020,155.848
C05046=1068.011,311.373,403.441,174.216,32.016,155.847
C05047=1068.005,311.125,403.474,174.212,32.012,155.846
C05048=1067.998,310.876,403.506,174.209,32.007,155.846
C05049=1067.992,310.629,403.539,174.206,32.003,155.845
C05050=1067.986,310.381,403.572,174.203,31.998,155.844
C05051=1067.979,310.133,403.603,174.199,31.994,155.843
C05052=1067.973,309.886,403.636,174.196,31.990,155.842
C05053=1067.967,309.638,403.668,174.194,31.985,155.841
C05054=1067.961,309.391,403.700,174.191,31.981,155.841
C05055=1067.955,309.143,403.733,174.188,31.977,155.840
C05056=1067.949,308.895,403.765,174.184,31.972,155.839
C05057=1067.943,308.647,403.798,174.181,31.968,155.838
C05058=1067.936,308.399,403.829,174.178,31.963,155.837
C05059=1067.930,308.152,403.862,174.175,31.959,155.836
C05060=1067.924,307.904,403.894,174.172,31.955,155.836
C05061=1067.917,307.656,403.927,174.169,31.950,155.835
C05062=1067.911,307.408,403.959,174.166,31.946,155.834
C05063=1067.905,307.160,403.992,174.163,31.942,155.833
C05064=1067.898,306.912,404.023,174.160,31.938,155.832
C05065=1067.893,306.665,404.055,174.156,31.933,155.832
C05066=1067.887,306.417,404.087,174.154,31.928,155.831
C05067=1067.881,306.169,404.119,174.151,31.924,155.830
C05068=1067.874,305.921,404.152,174.148,31.920,155.829
C05069=1067.868,305.673,404.184,174.145,31.916,155.828
C05070=1067.862,305.425,404.216,174.141,31.911,155.828
C05071=1067.856,305.178,404.248,174.138,31.907,155.827
C05072=1067.850,304.930,404.280,174.136,31.903,155.826
C05073=1067.844,304.701,404.309,174.133,31.898,155.825
C05074=1067.838,304.472,404.340,174.130,31.895,155.824
C05075=1067.833,304.243,404.369,174.127,31.890,155.824
C05076=1067.827,304.014,404.398,174.124,31.887,155.823
C05077=1067.821,303.785,404.428,174.121,31.882,155.822
C05078=1067.816,303.557,404.458,174.118,31.879,155.822
C05079=1067.810,303.328,404.487,174.116,31.874,155.821
C05080=1067.805,303.099,404.516,174.114,31.871,155.820
C05081=1067.799,302.851,404.548,174.110,31.866,155.819
C05082=1067.792,302.604,404.580,174.107,31.862,155.818
C05083=1067.786,302.356,404.612,174.104,31.857,155.818
C05084=1067.780,302.108,404.644,174.101,31.853,155.817
C05085=1067.775,301.860,404.676,174.099,31.849,155.816
C05086=1067.768,301.613,404.707,174.096,31.844,155.815
C05087=1067.762,301.364,404.739,174.093,31.840,155.814
C05088=1067.757,301.117,404.771,174.089,31.836,155.814
C05089=1067.750,300.869,404.802,174.086,31.831,155.813
C05090=1067.744,300.621,404.834,174.083,31.827,155.812
C05091=1067.739,300.373,404.866,174.081,31.823,155.811
C05092=1067.733,300.125,404.898,174.078,31.819,155.810
C05093=1067.726,299.877,404.929,174.075,31.814,155.810
C05094=1067.720,299.630,404.961,174.072,31.810,155.809
C05095=1067.714,299.381,404.993,174.069,31.806,155.808
C05096=1067.708,299.133,405.025,174.066,31.801,155.807
C05097=1067.702,298.886,405.056,174.063,31.797,155.806
C05098=1067.696,298.638,405.088,174.060,31.793,155.806
C05099=1067.690,298.391,405.119,174.057,31.788,155.805
C05100=1067.684,298.142,405.151,174.054,31.784,155.804
C05101=1067.678,297.894,405.183,174.051,31.780,155.803
C05102=1067.672,297.647,405.214,174.049,31.775,155.802
C05103=1067.666,297.399,405.246,174.046,31.771,155.802
C05104=1067.661,297.151,405.277,174.043,31.767,155.801
C05105=1067.654,296.903,405.309,174.040,31.763,155.800
C05106=1067.648,296.655,405.340,174.037,31.758,155.799
C05107=1067.642,296.407,405.372,174.033,31.754,155.799
C05108=1067.636,296.159,405.403,174.031,31.750,155.798
C05109=1067.630,295.911,405.434,174.028,31.746,155.797
C05110=1067.624,295.663,405.466,174.025,31.742,155.796
C05111=1067.617,295.415,405.497,174.022,31.737,155.795
C05112=1067.612,295.167,405.528,174.019,31.733,155.795
C05113=1067.605,294.919,405.560,174.017,31.729,155.794
C05114=1067.599,294.672,405.590,174.014,31.725,155.793
C05115=1067.593,294.423,405.622,174.011,31.721,155.792
C05116=1067.587,294.176,405.653,174.008,31.716,155.792
C05117=1067.581,293.928,405.684,174.005,31.713,155.791
C05118=1067.575,293.679,405.716,174.002,31.708,155.790
C05119=1067.569,293.432,405.746,174.000,31.704,155.789
C05120=1067.562,293.184,405.778,173.996,31.699,155.789
C05121=1067.556,292.936,405.809,173.993,31.696,155.788
C05122=1067.550,292.688,405.840,173.990,31.691,155.787
C05123=1067.544,292.440,405.871,173.987,31.687,155.786
C05124=1067.538,292.192,405.902,173.985,31.683,155.785
C05125=1067.533,291.944,405.933,173.982,31.679,155.785
C05126=1067.526,291.696,405.964,173.979,31.675,155.784
C05127=1067.520,291.448,405.994,173.976,31.670,155.783
C05128=1067.514,291.200,406.026,173.973,31.666,155.782
C05129=1067.509,290.978,406.054,173.971,31.662,155.782
C05130=1067.503,290.757,406.081,173.969,31.659,155.781
C05131=1067.497,290.536,406.108,173.966,31.655,155.780
C05132=1067.492,290.315,406.136,173.963,31.651,155.780
C05133=1067.487,290.093,406.164,173.961,31.648,155.779
C05134=1067.482,289.872,406.191,173.958,31.644,155.778
C05135=1067.476,289.651,406.218,173.956,31.640,155.778
C05136=1067.471,289.429,406.247,173.954,31.636,155.777
C05137=1067.464,289.181,406.278,173.951,31.633,155.776
C05138=1067.459,288.933,406.308,173.948,31.628,155.776
C05139=1067.453,288.686,406.339,173.945,31.624,155.775
C05140=1067.446,288.437,406.370,173.942,31.620,155.774
C05141=1067.440,288.189,406.400,173.939,31.616,155.773
C05142=1067.434,287.941,406.431,173.936,31.612,155.773
C05143=1067.428,287.694,406.462,173.933,31.608,155.772
C05144=1067.421,287.445,406.493,173.930,31.603,155.771
C05145=1067.416,287.197,406.523,173.927,31.600,155.770
C05146=1067.409,286.949,406.554,173.925,31.595,155.770
C05147=1067.403,286.701,406.584,173.922,31.592,155.769
C05148=1067.397,286.453,406.614,173.920,31.587,155.768
C05149=1067.391,286.205,406.645,173.917,31.583,155.767
C05150=1067.385,285.957,406.676,173.914,31.579,155.767
C05151=1067.379,285.709,406.707,173.912,31.575,155.766
C05152=1067.373,285.461,406.737,173.909,31.571,155.765
C05153=1067.367,285.213,406.767,173.906,31.567,155.764
C05154=1067.360,284.965,406.798,173.903,31.563,155.764
C05155=1067.355,284.717,406.829,173.900,31.559,155.763
C05156=1067.349,284.469,406.859,173.898,31.554,155.762
C05157=1067.342,284.221,406.890,173.895,31.551,155.761
C05158=1067.337,283.973,406.920,173.892,31.546,155.761
C05159=1067.331,283.725,406.950,173.889,31.542,155.760
C05160=1067.324,283.477,406.980,173.886,31.538,155.759
C05161=1067.318,283.229,407.011,173.884,31.534,155.758
C05162=1067.312,282.981,407.041,173.881,31.530,155.758
C05163=1067.306,282.732,407.071,173.878,31.526,155.757
C05164=1067.300,282.484,407.101,173.875,31.522,155.756
C05165=1067.294,282.236,407.132,173.873,31.518,155.756
C05166=1067.288,281.988,407.162,173.870,31.513,155.755
C05167=1067.282,281.740,407.193,173.867,31.509,155.754
C05168=1067.276,281.492,407.223,173.864,31.505,155.753
C05169=1067.270,281.244,407.254,173.861,31.501,155.752
C05170=1067.265,280.996,407.283,173.859,31.497,155.752
C05171=1067.258,280.747,407.314,173.857,31.493,155.751
C05172=1067.252,280.500,407.344,173.854,31.489,155.750
C05173=1067.246,280.252,407.374,173.851,31.485,155.750
C05174=1067.240,280.004,407.404,173.848,31.481,155.749
C05175=1067.234,279.755,407.434,173.846,31.477,155.748
C05176=1067.228,279.508,407.464,173.843,31.472,155.747
C05177=1067.222,279.260,407.495,173.840,31.469,155.747
C05178=1067.216,279.011,407.524,173.837,31.464,155.746
C05179=1067.209,278.763,407.554,173.834,31.461,155.745
C05180=1067.203,278.515,407.585,173.832,31.456,155.744
C05181=1067.198,278.267,407.614,173.829,31.452,155.744
C05182=1067.192,278.019,407.645,173.826,31.448,155.743
C05183=1067.185,277.770,407.674,173.824,31.444,155.742
C05184=1067.179,277.522,407.704,173.822,31.440,155.741
C05185=1067.174,277.307,407.731,173.819,31.437,155.741
C05186=1067.169,277.090,407.756,173.817,31.433,155.740
C05187=1067.164,276.874,407.783,173.814,31.429,155.740
C05188=1067.158,276.658,407.809,173.812,31.426,155.739
C05189=1067.153,276.441,407.834,173.810,31.423,155.738
C05190=1067.148,276.226,407.861,173.808,31.419,155.738
C05191=1067.142,276.009,407.887,173.805,31.416,155.737
C05192=1067.138,275.793,407.913,173.803,31.412,155.736
C05193=1067.131,275.545,407.942,173.800,31.408,155.736
C05194=1067.125,275.297,407.972,173.798,31.404,155.735
C05195=1067.119,275.048,408.002,173.795,31.400,155.734
C05196=1067.113,274.801,408.032,173.792,31.396,155.734
C05197=1067.107,274.552,408.062,173.789,31.392,155.733
C05198=1067.101,274.305,408.091,173.786,31.388,155.732
C05199=1067.095,274.056,408.121,173.784,31.384,155.731
C05200=1067.089,273.808,408.150,173.782,31.380,155.731
C05201=1067.083,273.560,408.180,173.779,31.376,155.730
C05202=1067.078,273.312,408.210,173.776,31.371,155.729
C05203=1067.071,273.064,408.239,173.774,31.368,155.728
C05204=1067.065,272.815,408.270,173.771,31.363,155.728
C05205=1067.059,272.567,408.299,173.768,31.359,155.727
C05206=1067.052,272.319,408.328,173.765,31.356,155.726
C05207=1067.047,272.071,408.357,173.763,31.351,155.726
C05208=1067.040,271.823,408.387,173.761,31.348,155.725
C05209=1067.035,271.598,408.413,173.758,31.344,155.724
C05210=1067.030,271.373,408.440,173.756,31.340,155.724
C05211=1067.025,271.149,408.467,173.753,31.336,155.723
C05212=1067.019,270.924,408.494,173.750,31.333,155.722
C05213=1067.014,270.698,408.521,173.749,31.330,155.722
C05214=1067.007,270.474,408.547,173.746,31.326,155.721
C05215=1067.002,270.249,408.574,173.744,31.322,155.720
C05216=1066.997,270.024,408.601,173.741,31.318,155.720
C05217=1066.991,269.776,408.630,173.739,31.314,155.719
C05218=1066.985,269.527,408.659,173.736,31.310,155.718
C05219=1066.979,269.280,408.689,173.734,31.306,155.718
C05220=1066.973,269.031,408.719,173.731,31.303,155.717
C05221=1066.967,268.783,408.748,173.728,31.298,155.716
C05222=1066.961,268.535,408.777,173.726,31.294,155.715
C05223=1066.954,268.287,408.806,173.723,31.290,155.715
C05224=1066.949,268.038,408.835,173.721,31.286,155.714
C05225=1066.943,267.790,408.864,173.718,31.283,155.713
C05226=1066.936,267.542,408.894,173.716,31.278,155.713
C05227=1066.931,267.294,408.923,173.713,31.274,155.712
C05228=1066.925,267.046,408.952,173.710,31.271,155.711
C05229=1066.918,266.797,408.981,173.708,31.266,155.710
C05230=1066.912,266.549,409.010,173.706,31.263,155.710
C05231=1066.907,266.301,409.040,173.703,31.258,155.709
C05232=1066.900,266.053,409.069,173.700,31.254,155.708
C05233=1066.894,265.805,409.098,173.697,31.251,155.708
C05234=1066.888,265.556,409.126,173.696,31.246,155.707
C05235=1066.883,265.307,409.156,173.693,31.243,155.706
C05236=1066.876,265.059,409.185,173.690,31.238,155.705
C05237=1066.870,264.811,409.214,173.687,31.234,155.705
C05238=1066.865,264.564,409.243,173.685,31.231,155.704
C05239=1066.858,264.316,409.272,173.683,31.226,155.703
C05240=1066.853,264.067,409.301,173.680,31.223,155.703
C05241=1066.847,263.829,409.329,173.677,31.219,155.702
C05242=1066.841,263.591,409.356,173.675,31.215,155.701
C05243=1066.835,263.354,409.384,173.673,31.211,155.701
C05244=1066.829,263.115,409.412,173.670,31.207,155.700
C05245=1066.823,262.878,409.440,173.668,31.204,155.699
C05246=1066.818,262.641,409.467,173.665,31.200,155.699
C05247=1066.812,262.402,409.494,173.663,31.196,155.698
C05248=1066.806,262.165,409.522,173.661,31.192,155.697
C05249=1066.800,261.916,409.551,173.658,31.188,155.696
C05250=1066.793,261.668,409.580,173.655,31.184,155.696
C05251=1066.787,261.420,409.609,173.653,31.180,155.695
C05252=1066.781,261.171,409.637,173.651,31.177,155.694
C05253=1066.774,260.923,409.665,173.648,31.172,155.694
C05254=1066.768,260.675,409.694,173.645,31.169,155.693
C05255=1066.762,260.427,409.723,173.643,31.165,155.692
C05256=1066.757,260.179,409.751,173.640,31.161,155.692
C05257=1066.750,259.930,409.780,173.638,31.157,155.691
C05258=1066.744,259.682,409.809,173.635,31.153,155.690
C05259=1066.738,259.434,409.837,173.633,31.149,155.690
C05260=1066.732,259.185,409.866,173.631,31.145,155.689
C05261=1066.726,258.937,409.894,173.628,31.141,155.688
C05262=1066.719,258.689,409.923,173.625,31.137,155.688
C05263=1066.713,258.440,409.951,173.623,31.133,155.687
C05264=1066.707,258.193,409.980,173.621,31.130,155.686
C05265=1066.702,257.944,410.008,173.618,31.125,155.685
C05266=1066.695,257.696,410.037,173.615,31.121,155.685
C05267=1066.689,257.447,410.066,173.613,31.118,155.684
C05268=1066.683,257.198,410.094,173.611,31.113,155.683
C05269=1066.677,256.951,410.122,173.608,31.109,155.683
C05270=1066.671,256.702,410.150,173.605,31.106,155.682
C05271=1066.665,256.454,410.179,173.604,31.101,155.681
C05272=1066.659,256.205,410.208,173.601,31.098,155.681
C05273=1066.653,255.957,410.236,173.598,31.094,155.680
C05274=1066.647,255.709,410.265,173.595,31.090,155.679
C05275=1066.641,255.461,410.292,173.594,31.086,155.678
C05276=1066.635,255.212,410.321,173.591,31.082,155.678
C05277=1066.628,254.964,410.350,173.588,31.078,155.677
C05278=1066.623,254.716,410.378,173.586,31.074,155.676
C05279=1066.617,254.467,410.406,173.584,31.070,155.676
C05280=1066.610,254.219,410.434,173.581,31.066,155.675
C05281=1066.605,253.971,410.462,173.579,31.062,155.674
C05282=1066.599,253.723,410.491,173.576,31.058,155.674
C05283=1066.593,253.474,410.519,173.574,31.054,155.673
C05284=1066.587,253.225,410.547,173.571,31.050,155.672
C05285=1066.581,252.977,410.575,173.569,31.046,155.671
C05286=1066.575,252.729,410.604,173.566,31.042,155.671
C05287=1066.569,252.480,410.632,173.564,31.038,155.670
C05288=1066.563,252.232,410.660,173.562,31.034,155.669
C05289=1066.557,251.984,410.688,173.559,31.030,155.669
C05290=1066.551,251.735,410.716,173.557,31.026,155.668
C05291=1066.545,251.487,410.744,173.555,31.022,155.667
C05292=1066.539,251.239,410.773,173.552,31.018,155.666
C05293=1066.534,250.991,410.801,173.549,31.014,155.666
C05294=1066.527,250.743,410.829,173.548,31.010,155.665
C05295=1066.521,250.494,410.857,173.545,31.006,155.664
C05296=1066.516,250.246,410.885,173.543,31.002,155.664
C05297=1066.510,250.030,410.910,173.540,30.998,155.663
C05298=1066.505,249.814,410.933,173.539,30.995,155.662
C05299=1066.500,249.599,410.958,173.537,30.992,155.662
C05300=1066.495,249.383,410.983,173.534,30.988,155.661
C05301=1066.491,249.168,411.007,173.532,30.985,155.661
C05302=1066.485,248.952,411.031,173.531,30.981,155.660
C05303=1066.480,248.737,411.055,173.529,30.978,155.659
C05304=1066.475,248.522,411.080,173.526,30.974,155.659
C05305=1066.469,248.272,411.107,173.524,30.970,155.658
C05306=1066.463,248.024,411.135,173.522,30.966,155.657
C05307=1066.457,247.776,411.163,173.519,30.962,155.657
C05308=1066.451,247.527,411.191,173.517,30.958,155.656
C05309=1066.446,247.279,411.219,173.514,30.954,155.655
C05310=1066.439,247.030,411.247,173.512,30.950,155.654
C05311=1066.434,246.782,411.275,173.510,30.946,155.654
C05312=1066.428,246.534,411.303,173.507,30.942,155.653
C05313=1066.422,246.286,411.331,173.506,30.938,155.652
C05314=1066.416,246.037,411.358,173.503,30.934,155.652
C05315=1066.410,245.789,411.386,173.500,30.930,155.651
C05316=1066.404,245.540,411.414,173.498,30.926,155.650
C05317=1066.398,245.292,411.441,173.496,30.922,155.649
C05318=1066.392,245.044,411.470,173.494,30.918,155.649
C05319=1066.387,244.795,411.496,173.491,30.914,155.648
C05320=1066.381,244.546,411.525,173.489,30.910,155.647
C05321=1066.374,244.299,411.552,173.487,30.906,155.647
C05322=1066.369,244.050,411.580,173.484,30.902,155.646
C05323=1066.363,243.802,411.607,173.482,30.898,155.645
C05324=1066.357,243.553,411.635,173.480,30.894,155.645
C05325=1066.351,243.305,411.663,173.477,30.890,155.644
C05326=1066.344,243.056,411.690,173.475,30.886,155.643
C05327=1066.339,242.808,411.718,173.472,30.882,155.643
C05328=1066.332,242.560,411.746,173.471,30.878,155.642
C05329=1066.327,242.311,411.773,173.468,30.874,155.641
C05330=1066.321,242.062,411.800,173.465,30.870,155.640
C05331=1066.315,241.814,411.827,173.464,30.866,155.640
C05332=1066.309,241.565,411.855,173.461,30.862,155.639
C05333=1066.303,241.318,411.883,173.459,30.858,155.638
C05334=1066.296,241.069,411.910,173.456,30.854,155.638
C05335=1066.290,240.821,411.937,173.455,30.850,155.637
C05336=1066.285,240.571,411.965,173.452,30.846,155.636
C05337=1066.279,240.324,411.992,173.449,30.842,155.636
C05338=1066.272,240.075,412.019,173.448,30.838,155.635
C05339=1066.266,239.827,412.047,173.445,30.834,155.634
C05340=1066.261,239.578,412.074,173.443,30.831,155.633
C05341=1066.254,239.330,412.102,173.441,30.826,155.633
C05342=1066.249,239.081,412.128,173.439,30.823,155.632
C05343=1066.242,238.832,412.155,173.436,30.819,155.631
C05344=1066.237,238.584,412.183,173.433,30.815,155.631
C05345=1066.231,238.335,412.210,173.432,30.811,155.630
C05346=1066.225,238.088,412.238,173.429,30.807,155.629
C05347=1066.218,237.838,412.265,173.427,30.803,155.629
C05348=1066.212,237.590,412.291,173.425,30.798,155.628
C05349=1066.206,237.342,412.319,173.423,30.795,155.627
C05350=1066.201,237.093,412.346,173.420,30.791,155.626
C05351=1066.195,236.845,412.373,173.418,30.787,155.626
C05352=1066.188,236.596,412.401,173.416,30.783,155.625
C05353=1066.183,236.378,412.424,173.414,30.779,155.624
C05354=1066.178,236.159,412.448,173.412,30.776,155.624
C05355=1066.173,235.940,412.472,173.410,30.772,155.623
C05356=1066.167,235.722,412.496,173.408,30.769,155.623
C05357=1066.163,235.503,412.519,173.406,30.765,155.622
C05358=1066.157,235.284,412.543,173.404,30.761,155.621
C05359=1066.152,235.066,412.567,173.402,30.758,155.621
C05360=1066.147,234.846,412.591,173.400,30.754,155.620
C05361=1066.141,234.598,412.618,173.398,30.751,155.619
C05362=1066.135,234.349,412.645,173.395,30.746,155.619
C05363=1066.129,234.101,412.672,173.394,30.743,155.618
C05364=1066.123,233.853,412.699,173.391,30.739,155.617
C05365=1066.116,233.604,412.726,173.389,30.734,155.617
C05366=1066.111,233.355,412.753,173.387,30.731,155.616
C05367=1066.106,233.107,412.779,173.385,30.727,155.615
C05368=1066.100,232.859,412.806,173.382,30.722,155.614
C05369=1066.093,232.610,412.834,173.381,30.719,155.614
C05370=1066.087,232.362,412.860,173.378,30.714,155.613
C05371=1066.082,232.113,412.887,173.376,30.711,155.612
C05372=1066.075,231.864,412.914,173.373,30.707,155.612
C05373=1066.069,231.616,412.941,173.372,30.702,155.611
C05374=1066.064,231.368,412.967,173.369,30.698,155.610
C05375=1066.058,231.119,412.994,173.367,30.695,155.610
C05376=1066.051,230.870,413.021,173.365,30.690,155.609
C05377=1066.046,230.622,413.048,173.363,30.687,155.608
C05378=1066.040,230.373,413.074,173.360,30.682,155.607
C05379=1066.034,230.125,413.101,173.359,30.678,155.607
C05380=1066.028,229.876,413.128,173.356,30.675,155.606
C05381=1066.021,229.628,413.154,173.354,30.670,155.605
C05382=1066.015,229.380,413.181,173.352,30.666,155.605
C05383=1066.010,229.131,413.207,173.350,30.663,155.604
C05384=1066.003,228.882,413.234,173.347,30.658,155.603
C05385=1065.998,228.634,413.261,173.346,30.654,155.603
C05386=1065.991,228.386,413.287,173.343,30.651,155.602
C05387=1065.986,228.137,413.313,173.341,30.646,155.601
C05388=1065.979,227.888,413.340,173.338,30.642,155.600
C05389=1065.973,227.639,413.367,173.337,30.639,155.600
C05390=1065.968,227.391,413.393,173.334,30.634,155.599
C05391=1065.961,227.143,413.419,173.332,30.631,155.598
C05392=1065.955,226.894,413.446,173.330,30.627,155.598
C05393=1065.949,226.646,413.473,173.328,30.622,155.597
C05394=1065.944,226.397,413.499,173.326,30.619,155.596
C05395=1065.937,226.148,413.525,173.324,30.615,155.596
C05396=1065.931,225.900,413.552,173.322,30.610,155.595
C05397=1065.925,225.652,413.578,173.319,30.607,155.594
C05398=1065.919,225.402,413.605,173.318,30.603,155.593
C05399=1065.913,225.154,413.631,173.315,30.598,155.593
C05400=1065.907,224.906,413.657,173.313,30.595,155.592
C05401=1065.901,224.657,413.684,173.311,30.590,155.591
C05402=1065.896,224.408,413.710,173.309,30.586,155.591
C05403=1065.889,224.160,413.736,173.307,30.583,155.590
C05404=1065.884,223.912,413.763,173.305,30.578,155.589
C05405=1065.878,223.662,413.789,173.303,30.574,155.589
C05406=1065.872,223.414,413.816,173.300,30.570,155.588
C05407=1065.865,223.166,413.842,173.299,30.566,155.587
C05408=1065.860,222.917,413.868,173.296,30.562,155.586
C05409=1065.854,222.695,413.891,173.294,30.559,155.586
C05410=1065.849,222.471,413.915,173.292,30.555,155.585
C05411=1065.844,222.249,413.938,173.291,30.551,155.584
C05412=1065.839,222.026,413.962,173.289,30.547,155.584
C05413=1065.833,221.803,413.986,173.287,30.544,155.583
C05414=1065.828,221.580,414.008,173.285,30.540,155.583
C05415=1065.823,221.358,414.032,173.283,30.537,155.582
C05416=1065.817,221.135,414.056,173.281,30.533,155.581
C05417=1065.811,220.886,414.082,173.280,30.529,155.581
C05418=1065.805,220.638,414.108,173.277,30.525,155.580
C05419=1065.799,220.389,414.134,173.275,30.521,155.579
C05420=1065.793,220.141,414.160,173.273,30.517,155.579
C05421=1065.787,219.892,414.186,173.271,30.513,155.578
C05422=1065.781,219.644,414.212,173.269,30.509,155.577
C05423=1065.775,219.395,414.237,173.267,30.505,155.576
C05424=1065.769,219.146,414.263,173.265,30.501,155.576
C05425=1065.763,218.898,414.289,173.262,30.497,155.575
C05426=1065.757,218.649,414.315,173.261,30.493,155.574
C05427=1065.751,218.401,414.341,173.259,30.489,155.574
C05428=1065.745,218.152,414.367,173.256,30.485,155.573
C05429=1065.739,217.904,414.393,173.255,30.481,155.572
C05430=1065.733,217.655,414.419,173.252,30.477,155.571
C05431=1065.727,217.407,414.445,173.250,30.473,155.571
C05432=1065.721,217.157,414.471,173.249,30.469,155.570
C05433=1065.715,216.909,414.497,173.246,30.465,155.569
C05434=1065.710,216.661,414.523,173.244,30.461,155.569
C05435=1065.703,216.412,414.548,173.242,30.457,155.568
C05436=1065.697,216.164,414.574,173.240,30.452,155.567
C05437=1065.691,215.915,414.600,173.238,30.449,155.567
C05438=1065.685,215.666,414.625,173.236,30.444,155.566
C05439=1065.680,215.418,414.652,173.234,30.440,155.565
C05440=1065.673,215.169,414.677,173.232,30.436,155.564
C05441=1065.668,214.920,414.703,173.230,30.432,155.564
C05442=1065.662,214.672,414.728,173.228,30.428,155.563
C05443=1065.655,214.423,414.754,173.225,30.424,155.562
C05444=1065.650,214.175,414.780,173.224,30.420,155.561
C05445=1065.643,213.926,414.806,173.222,30.416,155.561
C05446=1065.638,213.677,414.832,173.219,30.411,155.560
C05447=1065.632,213.428,414.857,173.218,30.408,155.559
C05448=1065.625,213.180,414.883,173.216,30.403,155.559
C05449=1065.620,212.931,414.909,173.214,30.399,155.558
C05450=1065.614,212.682,414.934,173.212,30.395,155.557
C05451=1065.608,212.435,414.959,173.210,30.391,155.556
C05452=1065.603,212.186,414.985,173.208,30.387,155.556
C05453=1065.596,211.937,415.011,173.206,30.383,155.555
C05454=1065.590,211.688,415.036,173.204,30.379,155.554
C05455=1065.585,211.439,415.062,173.202,30.375,155.554
C05456=1065.578,211.191,415.087,173.200,30.371,155.553
C05457=1065.572,210.942,415.113,173.198,30.367,155.552
C05458=1065.566,210.693,415.138,173.196,30.363,155.552
